LIN {X 0,Y 418.26,Z 369.386,A -85,B 0,C 180,E1 -10225.419,E2 -10225.419} C_VEL
LIN {X 0,Y 418.209,Z 369.388,A -85,B 0,C 180,E1 -10228.604,E2 -10228.604} C_VEL
LIN {X 0,Y 418.288,Z 369.379,A -85,B 0,C 180,E1 -10231.937,E2 -10231.937} C_VEL
LIN {X 0,Y 418.282,Z 369.366,A -85,B 0,C 180,E1 -10235.162,E2 -10235.162} C_VEL
LIN {X 0,Y 418.228,Z 369.385,A -85,B 0,C 180,E1 -10238.303,E2 -10238.303} C_VEL
LIN {X 0,Y 418.276,Z 369.382,A -85,B 0,C 180,E1 -10241.383,E2 -10241.383} C_VEL
LIN {X 0,Y 418.293,Z 369.376,A -85,B 0,C 180,E1 -10244.406,E2 -10244.406} C_VEL
LIN {X 0,Y 418.362,Z 369.372,A -85,B 0,C 180,E1 -10247.386,E2 -10247.386} C_VEL
LIN {X 0,Y 418.353,Z 369.367,A -85,B 0,C 180,E1 -10250.329,E2 -10250.329} C_VEL
LIN {X 0,Y 418.485,Z 369.352,A -85,B 0,C 180,E1 -10253.249,E2 -10253.249} C_VEL
LIN {X 0,Y 418.335,Z 369.376,A -85,B 0,C 180,E1 -10255.182,E2 -10255.182} C_VEL
LIN {X 0,Y 418.537,Z 369.345,A -85,B 0,C 180,E1 -10258.076,E2 -10258.076} C_VEL
LIN {X 0,Y 418.665,Z 369.329,A -85,B 0,C 180,E1 -10260,E2 -10260} C_VEL
LIN {X 0,Y 418.504,Z 369.351,A -85,B 0,C 180,E1 -10262.888,E2 -10262.888} C_VEL
LIN {X 0,Y 418.485,Z 369.357,A -85,B 0,C 180,E1 -10266.751,E2 -10266.751} C_VEL
LIN {X 0,Y 418.334,Z 369.372,A -85,B 0,C 180,E1 -10269.672,E2 -10269.672} C_VEL
LIN {X 0,Y 418.338,Z 369.373,A -85,B 0,C 180,E1 -10273.001,E2 -10273.001} C_VEL
LIN {X 0,Y 418.305,Z 369.376,A -85,B 0,C 180,E1 -10276.736,E2 -10276.736} C_VEL
LIN {X 0,Y 418.264,Z 369.382,A -85,B 0,C 180,E1 -10279.791,E2 -10279.791} C_VEL
LIN {X 0,Y 418.231,Z 369.389,A -85,B 0,C 180,E1 -10282.737,E2 -10282.737} C_VEL
LIN {X 0,Y 418.265,Z 369.372,A -85,B 0,C 180,E1 -10285.905,E2 -10285.905} C_VEL
LIN {X 0,Y 418.259,Z 369.382,A -85,B 0,C 180,E1 -10289.163,E2 -10289.163} C_VEL
LIN {X 0,Y 418.253,Z 369.384,A -85,B 0,C 180,E1 -10292.845,E2 -10292.845} C_VEL
LIN {X 0,Y 418.245,Z 369.388,A -85,B 0,C 180,E1 -10296.24,E2 -10296.24} C_VEL
LIN {X 0,Y 418.262,Z 369.384,A -85,B 0,C 180,E1 -10299.681,E2 -10299.681} C_VEL
LIN {X 0,Y 418.283,Z 369.379,A -85,B 0,C 180,E1 -10302.331,E2 -10302.331} C_VEL
LIN {X 0,Y 418.249,Z 369.388,A -85,B 0,C 180,E1 -10305.112,E2 -10305.112} C_VEL
LIN {X 0,Y 418.255,Z 369.391,A -85,B 0,C 180,E1 -10307.77,E2 -10307.77} C_VEL
LIN {X 0,Y 418.269,Z 369.384,A -85,B 0,C 180,E1 -10310.618,E2 -10310.618} C_VEL
LIN {X 0,Y 418.247,Z 369.387,A -85,B 0,C 180,E1 -10313.977,E2 -10313.977} C_VEL
LIN {X 0,Y 418.259,Z 369.385,A -85,B 0,C 180,E1 -10317.157,E2 -10317.157} C_VEL
LIN {X 0,Y 418.258,Z 369.391,A -85,B 0,C 180,E1 -10318.609,E2 -10318.609} C_VEL
LIN {X 0,Y 420.005,Z 378.049,A -85,B 0,C 180,E1 -10320.971,E2 -10320.971} C_VEL
LIN {X 0,Y 420.348,Z 380.959,A -85,B 0,C 180,E1 -10321.697,E2 -10321.697} C_VEL
LIN {X 0,Y 424.539,Z 397.902,A -85,B 0,C 180,E1 -10322.229,E2 -10322.229} C_VEL
LIN {X 0,Y 424.864,Z 400.946,A -85,B 0,C 180,E1 -10322.301,E2 -10322.301} C_VEL
LIN {X 0,Y 423.647,Z 487.611,A -85,B 0,C 180,E1 -10323.807,E2 -10323.807} C_VEL
LIN {X 0,Y 423.268,Z 499.777,A -85,B 0,C 180,E1 -10324.192,E2 -10324.192} C_VEL
LIN {X 0,Y 422.734,Z 512.426,A -85,B 0,C 180,E1 -10324.786,E2 -10324.786} C_VEL
LIN {X 0,Y 422.09,Z 524.174,A -85,B 0,C 180,E1 -10325.533,E2 -10325.533} C_VEL
LIN {X 0,Y 421.469,Z 534.802,A -85,B 0,C 180,E1 -10326.41,E2 -10326.41} C_VEL
LIN {X 0,Y 420.588,Z 545.68,A -85,B 0,C 180,E1 -10327.528,E2 -10327.528} C_VEL
LIN {X 0,Y 419.878,Z 554.518,A -85,B 0,C 180,E1 -10328.651,E2 -10328.651} C_VEL
LIN {X 0,Y 419.136,Z 563.264,A -85,B 0,C 180,E1 -10330.012,E2 -10330.012} C_VEL
LIN {X 0,Y 418.499,Z 570.426,A -85,B 0,C 180,E1 -10331.394,E2 -10331.394} C_VEL
LIN {X 0,Y 418.044,Z 576.652,A -85,B 0,C 180,E1 -10332.891,E2 -10332.891} C_VEL
LIN {X 0,Y 417.672,Z 581.55,A -85,B 0,C 180,E1 -10334.382,E2 -10334.382} C_VEL
LIN {X 0,Y 417.384,Z 585.282,A -85,B 0,C 180,E1 -10335.868,E2 -10335.868} C_VEL
LIN {X 0,Y 417.187,Z 588.485,A -85,B 0,C 180,E1 -10337.711,E2 -10337.711} C_VEL
LIN {X 0,Y 417.02,Z 590.19,A -85,B 0,C 180,E1 -10339.681,E2 -10339.681} C_VEL
LIN {X 0,Y 417.041,Z 590.444,A -85,B 0,C 180,E1 -10341.277,E2 -10341.277} C_VEL
LIN {X 0,Y 417.073,Z 590.067,A -85,B 0,C 180,E1 -10342.253,E2 -10342.253} C_VEL
LIN {X 0,Y 417.179,Z 588.496,A -85,B 0,C 180,E1 -10343.879,E2 -10343.879} C_VEL
LIN {X 0,Y 416.541,Z 587.399,A -85,B 0,C 180,E1 -10344.671,E2 -10344.671} C_VEL
LIN {X 0,Y 413.794,Z 585.076,A -85,B 0,C 180,E1 -10345.947,E2 -10345.947} C_VEL
LIN {X 0,Y 411.494,Z 582.788,A -85,B 0,C 180,E1 -10346.958,E2 -10346.958} C_VEL
LIN {X 0,Y 410.538,Z 580.679,A -85,B 0,C 180,E1 -10347.721,E2 -10347.721} C_VEL
LIN {X 0,Y 410.478,Z 579.858,A -85,B 0,C 180,E1 -10347.976,E2 -10347.976} C_VEL
LIN {X 0,Y 410.804,Z 574.307,A -85,B 0,C 180,E1 -10349.51,E2 -10349.51} C_VEL
LIN {X 0,Y 411.35,Z 567.599,A -85,B 0,C 180,E1 -10350.979,E2 -10350.979} C_VEL
LIN {X 0,Y 411.934,Z 559.285,A -85,B 0,C 180,E1 -10352.444,E2 -10352.444} C_VEL
LIN {X 0,Y 412.515,Z 550.731,A -85,B 0,C 180,E1 -10353.663,E2 -10353.663} C_VEL
LIN {X 0,Y 413.181,Z 540.216,A -85,B 0,C 180,E1 -10354.879,E2 -10354.879} C_VEL
LIN {X 0,Y 413.928,Z 529.748,A -85,B 0,C 180,E1 -10355.847,E2 -10355.847} C_VEL
LIN {X 0,Y 414.57,Z 518.155,A -85,B 0,C 180,E1 -10356.693,E2 -10356.693} C_VEL
LIN {X 0,Y 414.97,Z 506.184,A -85,B 0,C 180,E1 -10357.358,E2 -10357.358} C_VEL
LIN {X 0,Y 415.398,Z 493.099,A -85,B 0,C 180,E1 -10357.87,E2 -10357.87} C_VEL
LIN {X 0,Y 415.708,Z 480.345,A -85,B 0,C 180,E1 -10358.17,E2 -10358.17} C_VEL
LIN {X 0,Y 416.645,Z 399.493,A -85,B 0,C 180,E1 -10359.559,E2 -10359.559} C_VEL
LIN {X 0,Y 412.816,Z 380.72,A -85,B 0,C 180,E1 -10360.074,E2 -10360.074} C_VEL
LIN {X 0,Y 412.021,Z 373.906,A -85,B 0,C 180,E1 -10361.811,E2 -10361.811} C_VEL
LIN {X 0,Y 411.319,Z 370.252,A -85,B 0,C 180,E1 -10362.834,E2 -10362.834} C_VEL
LIN {X 0,Y 411.268,Z 370.259,A -85,B 0,C 180,E1 -10365.867,E2 -10365.867} C_VEL
LIN {X 0,Y 411.229,Z 370.259,A -85,B 0,C 180,E1 -10368.948,E2 -10368.948} C_VEL
LIN {X 0,Y 411.208,Z 370.263,A -85,B 0,C 180,E1 -10372.642,E2 -10372.642} C_VEL
LIN {X 0,Y 411.239,Z 370.256,A -85,B 0,C 180,E1 -10375.292,E2 -10375.292} C_VEL
LIN {X 0,Y 411.227,Z 370.261,A -85,B 0,C 180,E1 -10378.589,E2 -10378.589} C_VEL
LIN {X 0,Y 411.169,Z 370.268,A -85,B 0,C 180,E1 -10381.996,E2 -10381.996} C_VEL
LIN {X 0,Y 411.212,Z 370.262,A -85,B 0,C 180,E1 -10384.878,E2 -10384.878} C_VEL
LIN {X 0,Y 411.21,Z 370.265,A -85,B 0,C 180,E1 -10388.169,E2 -10388.169} C_VEL
LIN {X 0,Y 411.162,Z 370.267,A -85,B 0,C 180,E1 -10391.227,E2 -10391.227} C_VEL
LIN {X 0,Y 411.183,Z 370.267,A -85,B 0,C 180,E1 -10394.488,E2 -10394.488} C_VEL
LIN {X 0,Y 411.23,Z 370.258,A -85,B 0,C 180,E1 -10397.295,E2 -10397.295} C_VEL
LIN {X 0,Y 411.228,Z 370.261,A -85,B 0,C 180,E1 -10400.776,E2 -10400.776} C_VEL
LIN {X 0,Y 411.195,Z 370.265,A -85,B 0,C 180,E1 -10404.47,E2 -10404.47} C_VEL
LIN {X 0,Y 411.203,Z 370.263,A -85,B 0,C 180,E1 -10406.872,E2 -10406.872} C_VEL
LIN {X 0,Y 411.227,Z 370.261,A -85,B 0,C 180,E1 -10410.643,E2 -10410.643} C_VEL
LIN {X 0,Y 411.232,Z 370.259,A -85,B 0,C 180,E1 -10413.618,E2 -10413.618} C_VEL
LIN {X 0,Y 411.2,Z 370.263,A -85,B 0,C 180,E1 -10416.852,E2 -10416.852} C_VEL
LIN {X 0,Y 411.258,Z 370.258,A -85,B 0,C 180,E1 -10420.03,E2 -10420.03} C_VEL
LIN {X 0,Y 411.256,Z 370.256,A -85,B 0,C 180,E1 -10423.13,E2 -10423.13} C_VEL
LIN {X 0,Y 411.306,Z 370.25,A -85,B 0,C 180,E1 -10426.89,E2 -10426.89} C_VEL
LIN {X 0,Y 411.301,Z 370.252,A -85,B 0,C 180,E1 -10430.161,E2 -10430.161} C_VEL
LIN {X 0,Y 411.452,Z 370.231,A -85,B 0,C 180,E1 -10433.133,E2 -10433.133} C_VEL
LIN {X 0,Y 411.305,Z 370.249,A -85,B 0,C 180,E1 -10435.099,E2 -10435.099} C_VEL
LIN {X 0,Y 411.506,Z 370.227,A -85,B 0,C 180,E1 -10438.042,E2 -10438.042} C_VEL
LIN {X 0,Y 411.635,Z 370.211,A -85,B 0,C 180,E1 -10440,E2 -10440} C_VEL
LIN {X 0,Y 411.46,Z 370.23,A -85,B 0,C 180,E1 -10442.937,E2 -10442.937} C_VEL
LIN {X 0,Y 411.453,Z 370.231,A -85,B 0,C 180,E1 -10446.867,E2 -10446.867} C_VEL
LIN {X 0,Y 411.301,Z 370.252,A -85,B 0,C 180,E1 -10449.838,E2 -10449.838} C_VEL
LIN {X 0,Y 411.306,Z 370.249,A -85,B 0,C 180,E1 -10453.109,E2 -10453.109} C_VEL
LIN {X 0,Y 411.249,Z 370.256,A -85,B 0,C 180,E1 -10456.889,E2 -10456.889} C_VEL
LIN {X 0,Y 411.247,Z 370.259,A -85,B 0,C 180,E1 -10459.986,E2 -10459.986} C_VEL
LIN {X 0,Y 411.198,Z 370.262,A -85,B 0,C 180,E1 -10463.148,E2 -10463.148} C_VEL
LIN {X 0,Y 411.231,Z 370.261,A -85,B 0,C 180,E1 -10466.381,E2 -10466.381} C_VEL
LIN {X 0,Y 411.193,Z 370.265,A -85,B 0,C 180,E1 -10469.713,E2 -10469.713} C_VEL
LIN {X 0,Y 411.2,Z 370.262,A -85,B 0,C 180,E1 -10473.156,E2 -10473.156} C_VEL
LIN {X 0,Y 411.19,Z 370.264,A -85,B 0,C 180,E1 -10476.554,E2 -10476.554} C_VEL
LIN {X 0,Y 411.223,Z 370.262,A -85,B 0,C 180,E1 -10479.731,E2 -10479.731} C_VEL
LIN {X 0,Y 411.226,Z 370.258,A -85,B 0,C 180,E1 -10483.127,E2 -10483.127} C_VEL
LIN {X 0,Y 411.168,Z 370.27,A -85,B 0,C 180,E1 -10485.881,E2 -10485.881} C_VEL
LIN {X 0,Y 411.16,Z 370.266,A -85,B 0,C 180,E1 -10488.772,E2 -10488.772} C_VEL
LIN {X 0,Y 411.196,Z 370.266,A -85,B 0,C 180,E1 -10492.028,E2 -10492.028} C_VEL
LIN {X 0,Y 411.205,Z 370.264,A -85,B 0,C 180,E1 -10495.667,E2 -10495.667} C_VEL
LIN {X 0,Y 411.199,Z 370.262,A -85,B 0,C 180,E1 -10499.154,E2 -10499.154} C_VEL
LIN {X 0,Y 411.29,Z 370.439,A -85,B 0,C 180,E1 -10501.834,E2 -10501.834} C_VEL
LIN {X 0,Y 413.861,Z 383.381,A -85,B 0,C 180,E1 -10504.573,E2 -10504.573} C_VEL
LIN {X 0,Y 414.249,Z 387.672,A -85,B 0,C 180,E1 -10505.44,E2 -10505.44} C_VEL
LIN {X 0,Y 413.21,Z 403.81,A -85,B 0,C 180,E1 -10508.551,E2 -10508.551} C_VEL
LIN {X 0,Y 412.423,Z 416.273,A -85,B 0,C 180,E1 -10510.934,E2 -10510.934} C_VEL
LIN {X 0,Y 416.349,Z 445.438,A -85,B 0,C 180,E1 -10511.607,E2 -10511.607} C_VEL
LIN {X 0,Y 415.451,Z 525.237,A -85,B 0,C 180,E1 -10513.002,E2 -10513.002} C_VEL
LIN {X 0,Y 414.843,Z 539.187,A -85,B 0,C 180,E1 -10513.452,E2 -10513.452} C_VEL
LIN {X 0,Y 414.285,Z 551.698,A -85,B 0,C 180,E1 -10514.062,E2 -10514.062} C_VEL
LIN {X 0,Y 413.532,Z 563.64,A -85,B 0,C 180,E1 -10514.853,E2 -10514.853} C_VEL
LIN {X 0,Y 412.761,Z 575.122,A -85,B 0,C 180,E1 -10515.833,E2 -10515.833} C_VEL
LIN {X 0,Y 412.124,Z 585.675,A -85,B 0,C 180,E1 -10516.965,E2 -10516.965} C_VEL
LIN {X 0,Y 411.501,Z 594.764,A -85,B 0,C 180,E1 -10518.174,E2 -10518.174} C_VEL
LIN {X 0,Y 410.818,Z 603.786,A -85,B 0,C 180,E1 -10519.652,E2 -10519.652} C_VEL
LIN {X 0,Y 410.456,Z 611.054,A -85,B 0,C 180,E1 -10521.136,E2 -10521.136} C_VEL
LIN {X 0,Y 410.183,Z 616.842,A -85,B 0,C 180,E1 -10522.617,E2 -10522.617} C_VEL
LIN {X 0,Y 410.007,Z 621.393,A -85,B 0,C 180,E1 -10524.097,E2 -10524.097} C_VEL
LIN {X 0,Y 410.047,Z 623.795,A -85,B 0,C 180,E1 -10525.084,E2 -10525.084} C_VEL
LIN {X 0,Y 409.954,Z 625.753,A -85,B 0,C 180,E1 -10526.068,E2 -10526.068} C_VEL
LIN {X 0,Y 410.007,Z 627.296,A -85,B 0,C 180,E1 -10527.052,E2 -10527.052} C_VEL
LIN {X 0,Y 410.021,Z 628.38,A -85,B 0,C 180,E1 -10528.035,E2 -10528.035} C_VEL
LIN {X 0,Y 409.972,Z 629.348,A -85,B 0,C 180,E1 -10530,E2 -10530} C_VEL
LIN {X 0,Y 409.978,Z 629.25,A -85,B 0,C 180,E1 -10530.982,E2 -10530.982} C_VEL
LIN {X 0,Y 410.018,Z 628.721,A -85,B 0,C 180,E1 -10531.965,E2 -10531.965} C_VEL
LIN {X 0,Y 409.97,Z 627.786,A -85,B 0,C 180,E1 -10532.948,E2 -10532.948} C_VEL
LIN {X 0,Y 410.024,Z 624.725,A -85,B 0,C 180,E1 -10534.916,E2 -10534.916} C_VEL
LIN {X 0,Y 410.041,Z 621.689,A -85,B 0,C 180,E1 -10536.224,E2 -10536.224} C_VEL
LIN {X 0,Y 410.285,Z 616.703,A -85,B 0,C 180,E1 -10537.876,E2 -10537.876} C_VEL
LIN {X 0,Y 410.705,Z 609.834,A -85,B 0,C 180,E1 -10539.604,E2 -10539.604} C_VEL
LIN {X 0,Y 411.27,Z 602.404,A -85,B 0,C 180,E1 -10541.084,E2 -10541.084} C_VEL
LIN {X 0,Y 412.095,Z 593.192,A -85,B 0,C 180,E1 -10542.559,E2 -10542.559} C_VEL
LIN {X 0,Y 412.78,Z 583.641,A -85,B 0,C 180,E1 -10543.79,E2 -10543.79} C_VEL
LIN {X 0,Y 413.627,Z 573.075,A -85,B 0,C 180,E1 -10544.891,E2 -10544.891} C_VEL
LIN {X 0,Y 414.603,Z 561.291,A -85,B 0,C 180,E1 -10545.863,E2 -10545.863} C_VEL
LIN {X 0,Y 415.447,Z 548.69,A -85,B 0,C 180,E1 -10546.65,E2 -10546.65} C_VEL
LIN {X 0,Y 416.229,Z 535.368,A -85,B 0,C 180,E1 -10547.25,E2 -10547.25} C_VEL
LIN {X 0,Y 416.706,Z 523.005,A -85,B 0,C 180,E1 -10547.609,E2 -10547.609} C_VEL
LIN {X 0,Y 417.673,Z 444.319,A -85,B 0,C 180,E1 -10548.995,E2 -10548.995} C_VEL
LIN {X 0,Y 413.987,Z 421.068,A -85,B 0,C 180,E1 -10549.618,E2 -10549.618} C_VEL
LIN {X 0,Y 413.043,Z 415.819,A -85,B 0,C 180,E1 -10549.791,E2 -10549.791} C_VEL
LIN {X 0,Y 414.399,Z 397.757,A -85,B 0,C 180,E1 -10553.343,E2 -10553.343} C_VEL
LIN {X 0,Y 415.069,Z 389.228,A -85,B 0,C 180,E1 -10555.043,E2 -10555.043} C_VEL
LIN {X 0,Y 413.772,Z 381.411,A -85,B 0,C 180,E1 -10556.75,E2 -10556.75} C_VEL
LIN {X 0,Y 411.233,Z 370.258,A -85,B 0,C 180,E1 -10559.321,E2 -10559.321} C_VEL
LIN {X 0,Y 411.206,Z 370.263,A -85,B 0,C 180,E1 -10563.126,E2 -10563.126} C_VEL
LIN {X 0,Y 411.193,Z 370.265,A -85,B 0,C 180,E1 -10566.552,E2 -10566.552} C_VEL
LIN {X 0,Y 411.215,Z 370.263,A -85,B 0,C 180,E1 -10569.728,E2 -10569.728} C_VEL
LIN {X 0,Y 411.169,Z 370.264,A -85,B 0,C 180,E1 -10573.133,E2 -10573.133} C_VEL
LIN {X 0,Y 411.228,Z 370.259,A -85,B 0,C 180,E1 -10575.871,E2 -10575.871} C_VEL
LIN {X 0,Y 411.205,Z 370.257,A -85,B 0,C 180,E1 -10578.764,E2 -10578.764} C_VEL
LIN {X 0,Y 411.198,Z 370.261,A -85,B 0,C 180,E1 -10582.027,E2 -10582.027} C_VEL
LIN {X 0,Y 411.2,Z 370.265,A -85,B 0,C 180,E1 -10585.666,E2 -10585.666} C_VEL
LIN {X 0,Y 411.191,Z 370.266,A -85,B 0,C 180,E1 -10589.153,E2 -10589.153} C_VEL
LIN {X 0,Y 411.253,Z 370.254,A -85,B 0,C 180,E1 -10592.522,E2 -10592.522} C_VEL
LIN {X 0,Y 411.22,Z 370.249,A -85,B 0,C 180,E1 -10595.784,E2 -10595.784} C_VEL
LIN {X 0,Y 411.19,Z 370.265,A -85,B 0,C 180,E1 -10598.966,E2 -10598.966} C_VEL
LIN {X 0,Y 411.244,Z 370.255,A -85,B 0,C 180,E1 -10602.085,E2 -10602.085} C_VEL
LIN {X 0,Y 411.254,Z 370.254,A -85,B 0,C 180,E1 -10605.147,E2 -10605.147} C_VEL
LIN {X 0,Y 411.292,Z 370.249,A -85,B 0,C 180,E1 -10608.168,E2 -10608.168} C_VEL
LIN {X 0,Y 411.473,Z 370.227,A -85,B 0,C 180,E1 -10612.147,E2 -10612.147} C_VEL
LIN {X 0,Y 411.467,Z 370.222,A -85,B 0,C 180,E1 -10614.118,E2 -10614.118} C_VEL
LIN {X 0,Y 411.506,Z 370.221,A -85,B 0,C 180,E1 -10618.043,E2 -10618.043} C_VEL
LIN {X 0,Y 411.635,Z 370.205,A -85,B 0,C 180,E1 -10620,E2 -10620} C_VEL
LIN {X 0,Y 411.459,Z 370.228,A -85,B 0,C 180,E1 -10622.938,E2 -10622.938} C_VEL
LIN {X 0,Y 411.452,Z 370.231,A -85,B 0,C 180,E1 -10626.867,E2 -10626.867} C_VEL
LIN {X 0,Y 411.286,Z 370.25,A -85,B 0,C 180,E1 -10629.839,E2 -10629.839} C_VEL
LIN {X 0,Y 411.298,Z 370.249,A -85,B 0,C 180,E1 -10633.105,E2 -10633.105} C_VEL
LIN {X 0,Y 411.256,Z 370.254,A -85,B 0,C 180,E1 -10636.87,E2 -10636.87} C_VEL
LIN {X 0,Y 411.224,Z 370.26,A -85,B 0,C 180,E1 -10639.988,E2 -10639.988} C_VEL
LIN {X 0,Y 411.197,Z 370.262,A -85,B 0,C 180,E1 -10643.148,E2 -10643.148} C_VEL
LIN {X 0,Y 411.232,Z 370.245,A -85,B 0,C 180,E1 -10646.382,E2 -10646.382} C_VEL
LIN {X 0,Y 411.195,Z 370.263,A -85,B 0,C 180,E1 -10649.714,E2 -10649.714} C_VEL
LIN {X 0,Y 411.202,Z 370.261,A -85,B 0,C 180,E1 -10653.157,E2 -10653.157} C_VEL
LIN {X 0,Y 411.192,Z 370.264,A -85,B 0,C 180,E1 -10656.554,E2 -10656.554} C_VEL
LIN {X 0,Y 411.224,Z 370.262,A -85,B 0,C 180,E1 -10659.731,E2 -10659.731} C_VEL
LIN {X 0,Y 411.222,Z 370.259,A -85,B 0,C 180,E1 -10663.128,E2 -10663.128} C_VEL
LIN {X 0,Y 411.17,Z 370.269,A -85,B 0,C 180,E1 -10665.882,E2 -10665.882} C_VEL
LIN {X 0,Y 411.212,Z 370.267,A -85,B 0,C 180,E1 -10669.501,E2 -10669.501} C_VEL
LIN {X 0,Y 411.205,Z 370.266,A -85,B 0,C 180,E1 -10672.029,E2 -10672.029} C_VEL
LIN {X 0,Y 411.207,Z 370.264,A -85,B 0,C 180,E1 -10675.668,E2 -10675.668} C_VEL
LIN {X 0,Y 411.243,Z 370.437,A -85,B 0,C 180,E1 -10678.347,E2 -10678.347} C_VEL
LIN {X 0,Y 413.074,Z 379.492,A -85,B 0,C 180,E1 -10680.858,E2 -10680.858} C_VEL
LIN {X 0,Y 413.38,Z 381.416,A -85,B 0,C 180,E1 -10681.311,E2 -10681.311} C_VEL
LIN {X 0,Y 416.742,Z 393.57,A -85,B 0,C 180,E1 -10681.726,E2 -10681.726} C_VEL
LIN {X 0,Y 418.272,Z 401.497,A -85,B 0,C 180,E1 -10681.955,E2 -10681.955} C_VEL
LIN {X 0,Y 416.976,Z 487.866,A -85,B 0,C 180,E1 -10683.478,E2 -10683.478} C_VEL
LIN {X 0,Y 416.542,Z 500.63,A -85,B 0,C 180,E1 -10683.891,E2 -10683.891} C_VEL
LIN {X 0,Y 416.009,Z 512.932,A -85,B 0,C 180,E1 -10684.483,E2 -10684.483} C_VEL
LIN {X 0,Y 415.331,Z 524.629,A -85,B 0,C 180,E1 -10685.241,E2 -10685.241} C_VEL
LIN {X 0,Y 414.667,Z 535.319,A -85,B 0,C 180,E1 -10686.141,E2 -10686.141} C_VEL
LIN {X 0,Y 413.749,Z 546.088,A -85,B 0,C 180,E1 -10687.268,E2 -10687.268} C_VEL
LIN {X 0,Y 412.937,Z 555.815,A -85,B 0,C 180,E1 -10688.536,E2 -10688.536} C_VEL
LIN {X 0,Y 412.213,Z 563.693,A -85,B 0,C 180,E1 -10689.801,E2 -10689.801} C_VEL
LIN {X 0,Y 411.492,Z 571.362,A -85,B 0,C 180,E1 -10691.323,E2 -10691.323} C_VEL
LIN {X 0,Y 410.938,Z 578.382,A -85,B 0,C 180,E1 -10693.098,E2 -10693.098} C_VEL
LIN {X 0,Y 410.553,Z 582.966,A -85,B 0,C 180,E1 -10694.614,E2 -10694.614} C_VEL
LIN {X 0,Y 410.288,Z 586.419,A -85,B 0,C 180,E1 -10696.125,E2 -10696.125} C_VEL
LIN {X 0,Y 410.131,Z 588.831,A -85,B 0,C 180,E1 -10697.624,E2 -10697.624} C_VEL
LIN {X 0,Y 409.994,Z 590.297,A -85,B 0,C 180,E1 -10699.132,E2 -10699.132} C_VEL
LIN {X 0,Y 409.909,Z 590.756,A -85,B 0,C 180,E1 -10700.128,E2 -10700.128} C_VEL
LIN {X 0,Y 409.976,Z 590.459,A -85,B 0,C 180,E1 -10702.118,E2 -10702.118} C_VEL
LIN {X 0,Y 410.091,Z 588.842,A -85,B 0,C 180,E1 -10703.889,E2 -10703.889} C_VEL
LIN {X 0,Y 410.12,Z 587.009,A -85,B 0,C 180,E1 -10705.085,E2 -10705.085} C_VEL
LIN {X 0,Y 410.329,Z 583.857,A -85,B 0,C 180,E1 -10706.563,E2 -10706.563} C_VEL
LIN {X 0,Y 410.478,Z 579.858,A -85,B 0,C 180,E1 -10707.976,E2 -10707.976} C_VEL
LIN {X 0,Y 409.915,Z 577.429,A -85,B 0,C 180,E1 -10708.726,E2 -10708.726} C_VEL
LIN {X 0,Y 407.36,Z 573.051,A -85,B 0,C 180,E1 -10709.924,E2 -10709.924} C_VEL
LIN {X 0,Y 404.927,Z 568.02,A -85,B 0,C 180,E1 -10711.082,E2 -10711.082} C_VEL
LIN {X 0,Y 404.556,Z 564.541,A -85,B 0,C 180,E1 -10711.758,E2 -10711.758} C_VEL
LIN {X 0,Y 405.245,Z 555.484,A -85,B 0,C 180,E1 -10713.231,E2 -10713.231} C_VEL
LIN {X 0,Y 405.972,Z 544.95,A -85,B 0,C 180,E1 -10714.592,E2 -10714.592} C_VEL
LIN {X 0,Y 406.736,Z 534.195,A -85,B 0,C 180,E1 -10715.702,E2 -10715.702} C_VEL
LIN {X 0,Y 407.404,Z 523.685,A -85,B 0,C 180,E1 -10716.562,E2 -10716.562} C_VEL
LIN {X 0,Y 407.922,Z 511.113,A -85,B 0,C 180,E1 -10717.362,E2 -10717.362} C_VEL
LIN {X 0,Y 408.397,Z 498.485,A -85,B 0,C 180,E1 -10717.944,E2 -10717.944} C_VEL
LIN {X 0,Y 408.737,Z 486.317,A -85,B 0,C 180,E1 -10718.31,E2 -10718.31} C_VEL
LIN {X 0,Y 409.873,Z 400.613,A -85,B 0,C 180,E1 -10719.818,E2 -10719.818} C_VEL
LIN {X 0,Y 405.82,Z 381.046,A -85,B 0,C 180,E1 -10720.364,E2 -10720.364} C_VEL
LIN {X 0,Y 404.625,Z 372.722,A -85,B 0,C 180,E1 -10722.539,E2 -10722.539} C_VEL
LIN {X 0,Y 404.277,Z 371.129,A -85,B 0,C 180,E1 -10722.997,E2 -10722.997} C_VEL
LIN {X 0,Y 404.232,Z 371.135,A -85,B 0,C 180,E1 -10726.151,E2 -10726.151} C_VEL
LIN {X 0,Y 404.17,Z 371.137,A -85,B 0,C 180,E1 -10729.292,E2 -10729.292} C_VEL
LIN {X 0,Y 404.159,Z 371.14,A -85,B 0,C 180,E1 -10732.833,E2 -10732.833} C_VEL
LIN {X 0,Y 404.187,Z 371.135,A -85,B 0,C 180,E1 -10735.766,E2 -10735.766} C_VEL
LIN {X 0,Y 404.201,Z 371.135,A -85,B 0,C 180,E1 -10737.999,E2 -10737.999} C_VEL
LIN {X 0,Y 404.144,Z 371.14,A -85,B 0,C 180,E1 -10741.558,E2 -10741.558} C_VEL
LIN {X 0,Y 404.186,Z 371.136,A -85,B 0,C 180,E1 -10745.015,E2 -10745.015} C_VEL
LIN {X 0,Y 404.157,Z 371.141,A -85,B 0,C 180,E1 -10748.756,E2 -10748.756} C_VEL
LIN {X 0,Y 404.121,Z 371.144,A -85,B 0,C 180,E1 -10751.599,E2 -10751.599} C_VEL
LIN {X 0,Y 404.151,Z 371.143,A -85,B 0,C 180,E1 -10754.522,E2 -10754.522} C_VEL
LIN {X 0,Y 404.208,Z 371.133,A -85,B 0,C 180,E1 -10757.304,E2 -10757.304} C_VEL
LIN {X 0,Y 404.166,Z 371.141,A -85,B 0,C 180,E1 -10759.954,E2 -10759.954} C_VEL
LIN {X 0,Y 404.137,Z 371.142,A -85,B 0,C 180,E1 -10763.123,E2 -10763.123} C_VEL
LIN {X 0,Y 404.141,Z 371.145,A -85,B 0,C 180,E1 -10766.187,E2 -10766.187} C_VEL
LIN {X 0,Y 404.14,Z 371.143,A -85,B 0,C 180,E1 -10769.714,E2 -10769.714} C_VEL
LIN {X 0,Y 404.19,Z 371.135,A -85,B 0,C 180,E1 -10773.122,E2 -10773.122} C_VEL
LIN {X 0,Y 404.165,Z 371.141,A -85,B 0,C 180,E1 -10776.425,E2 -10776.425} C_VEL
LIN {X 0,Y 404.199,Z 371.138,A -85,B 0,C 180,E1 -10779.868,E2 -10779.868} C_VEL
LIN {X 0,Y 404.209,Z 371.133,A -85,B 0,C 180,E1 -10782.992,E2 -10782.992} C_VEL
LIN {X 0,Y 404.259,Z 371.128,A -85,B 0,C 180,E1 -10786.788,E2 -10786.788} C_VEL
LIN {X 0,Y 404.264,Z 371.129,A -85,B 0,C 180,E1 -10789.988,E2 -10789.988} C_VEL
LIN {X 0,Y 404.403,Z 371.109,A -85,B 0,C 180,E1 -10793.012,E2 -10793.012} C_VEL
LIN {X 0,Y 404.277,Z 371.125,A -85,B 0,C 180,E1 -10795.013,E2 -10795.013} C_VEL
LIN {X 0,Y 404.475,Z 371.103,A -85,B 0,C 180,E1 -10798.008,E2 -10798.008} C_VEL
LIN {X 0,Y 404.605,Z 371.087,A -85,B 0,C 180,E1 -10800,E2 -10800} C_VEL
LIN {X 0,Y 404.417,Z 371.107,A -85,B 0,C 180,E1 -10802.988,E2 -10802.988} C_VEL
LIN {X 0,Y 404.404,Z 371.109,A -85,B 0,C 180,E1 -10806.987,E2 -10806.987} C_VEL
LIN {X 0,Y 404.264,Z 371.129,A -85,B 0,C 180,E1 -10810.011,E2 -10810.011} C_VEL
LIN {X 0,Y 404.258,Z 371.127,A -85,B 0,C 180,E1 -10813.211,E2 -10813.211} C_VEL
LIN {X 0,Y 404.208,Z 371.133,A -85,B 0,C 180,E1 -10817.007,E2 -10817.007} C_VEL
LIN {X 0,Y 404.193,Z 371.138,A -85,B 0,C 180,E1 -10820.35,E2 -10820.35} C_VEL
LIN {X 0,Y 404.164,Z 371.141,A -85,B 0,C 180,E1 -10823.575,E2 -10823.575} C_VEL
LIN {X 0,Y 404.188,Z 371.135,A -85,B 0,C 180,E1 -10826.878,E2 -10826.878} C_VEL
LIN {X 0,Y 404.138,Z 371.145,A -85,B 0,C 180,E1 -10830.286,E2 -10830.286} C_VEL
LIN {X 0,Y 404.139,Z 371.145,A -85,B 0,C 180,E1 -10833.813,E2 -10833.813} C_VEL
LIN {X 0,Y 404.135,Z 371.142,A -85,B 0,C 180,E1 -10836.876,E2 -10836.876} C_VEL
LIN {X 0,Y 404.163,Z 371.143,A -85,B 0,C 180,E1 -10840.084,E2 -10840.084} C_VEL
LIN {X 0,Y 404.2,Z 371.133,A -85,B 0,C 180,E1 -10843.092,E2 -10843.092} C_VEL
LIN {X 0,Y 404.147,Z 371.145,A -85,B 0,C 180,E1 -10845.927,E2 -10845.927} C_VEL
LIN {X 0,Y 404.114,Z 371.144,A -85,B 0,C 180,E1 -10848.636,E2 -10848.636} C_VEL
LIN {X 0,Y 404.153,Z 371.141,A -85,B 0,C 180,E1 -10851.492,E2 -10851.492} C_VEL
LIN {X 0,Y 404.183,Z 371.135,A -85,B 0,C 180,E1 -10854.985,E2 -10854.985} C_VEL
LIN {X 0,Y 404.148,Z 371.139,A -85,B 0,C 180,E1 -10858.555,E2 -10858.555} C_VEL
LIN {X 0,Y 404.238,Z 371.226,A -85,B 0,C 180,E1 -10861.58,E2 -10861.58} C_VEL
LIN {X 0,Y 406.506,Z 382.537,A -85,B 0,C 180,E1 -10864.029,E2 -10864.029} C_VEL
LIN {X 0,Y 407.304,Z 388.468,A -85,B 0,C 180,E1 -10865.265,E2 -10865.265} C_VEL
LIN {X 0,Y 406.207,Z 404.596,A -85,B 0,C 180,E1 -10868.429,E2 -10868.429} C_VEL
LIN {X 0,Y 405.462,Z 415.961,A -85,B 0,C 180,E1 -10870.641,E2 -10870.641} C_VEL
LIN {X 0,Y 409.518,Z 445.084,A -85,B 0,C 180,E1 -10871.332,E2 -10871.332} C_VEL
LIN {X 0,Y 408.595,Z 524.516,A -85,B 0,C 180,E1 -10872.74,E2 -10872.74} C_VEL
LIN {X 0,Y 408.044,Z 537.839,A -85,B 0,C 180,E1 -10873.168,E2 -10873.168} C_VEL
LIN {X 0,Y 407.415,Z 550.633,A -85,B 0,C 180,E1 -10873.786,E2 -10873.786} C_VEL
LIN {X 0,Y 406.661,Z 562.784,A -85,B 0,C 180,E1 -10874.591,E2 -10874.591} C_VEL
LIN {X 0,Y 405.807,Z 574.358,A -85,B 0,C 180,E1 -10875.585,E2 -10875.585} C_VEL
LIN {X 0,Y 405.153,Z 585.264,A -85,B 0,C 180,E1 -10876.769,E2 -10876.769} C_VEL
LIN {X 0,Y 404.522,Z 594.164,A -85,B 0,C 180,E1 -10877.967,E2 -10877.967} C_VEL
LIN {X 0,Y 403.793,Z 603.232,A -85,B 0,C 180,E1 -10879.47,E2 -10879.47} C_VEL
LIN {X 0,Y 403.379,Z 610.541,A -85,B 0,C 180,E1 -10880.979,E2 -10880.979} C_VEL
LIN {X 0,Y 403.129,Z 616.378,A -85,B 0,C 180,E1 -10882.487,E2 -10882.487} C_VEL
LIN {X 0,Y 402.938,Z 620.961,A -85,B 0,C 180,E1 -10883.993,E2 -10883.993} C_VEL
LIN {X 0,Y 402.954,Z 623.378,A -85,B 0,C 180,E1 -10884.997,E2 -10884.997} C_VEL
LIN {X 0,Y 402.874,Z 625.35,A -85,B 0,C 180,E1 -10885.999,E2 -10885.999} C_VEL
LIN {X 0,Y 402.906,Z 626.909,A -85,B 0,C 180,E1 -10887,E2 -10887} C_VEL
LIN {X 0,Y 402.951,Z 628.016,A -85,B 0,C 180,E1 -10888.001,E2 -10888.001} C_VEL
LIN {X 0,Y 402.894,Z 629.008,A -85,B 0,C 180,E1 -10890,E2 -10890} C_VEL
LIN {X 0,Y 402.903,Z 628.924,A -85,B 0,C 180,E1 -10890.999,E2 -10890.999} C_VEL
LIN {X 0,Y 402.946,Z 628.419,A -85,B 0,C 180,E1 -10891.999,E2 -10891.999} C_VEL
LIN {X 0,Y 402.861,Z 626.179,A -85,B 0,C 180,E1 -10894.001,E2 -10894.001} C_VEL
LIN {X 0,Y 402.92,Z 623.404,A -85,B 0,C 180,E1 -10895.505,E2 -10895.505} C_VEL
LIN {X 0,Y 403.076,Z 619.614,A -85,B 0,C 180,E1 -10897.01,E2 -10897.01} C_VEL
LIN {X 0,Y 403.328,Z 614.712,A -85,B 0,C 180,E1 -10898.517,E2 -10898.517} C_VEL
LIN {X 0,Y 403.746,Z 608.555,A -85,B 0,C 180,E1 -10900.024,E2 -10900.024} C_VEL
LIN {X 0,Y 404.387,Z 600.926,A -85,B 0,C 180,E1 -10901.529,E2 -10901.529} C_VEL
LIN {X 0,Y 405.156,Z 593.143,A -85,B 0,C 180,E1 -10902.777,E2 -10902.777} C_VEL
LIN {X 0,Y 405.862,Z 583.662,A -85,B 0,C 180,E1 -10904.03,E2 -10904.03} C_VEL
LIN {X 0,Y 406.78,Z 573.173,A -85,B 0,C 180,E1 -10905.148,E2 -10905.148} C_VEL
LIN {X 0,Y 407.77,Z 561.524,A -85,B 0,C 180,E1 -10906.136,E2 -10906.136} C_VEL
LIN {X 0,Y 408.687,Z 549.117,A -85,B 0,C 180,E1 -10906.933,E2 -10906.933} C_VEL
LIN {X 0,Y 409.482,Z 536.076,A -85,B 0,C 180,E1 -10907.543,E2 -10907.543} C_VEL
LIN {X 0,Y 410.017,Z 523.226,A -85,B 0,C 180,E1 -10907.938,E2 -10907.938} C_VEL
LIN {X 0,Y 410.998,Z 444.67,A -85,B 0,C 180,E1 -10909.349,E2 -10909.349} C_VEL
LIN {X 0,Y 407.41,Z 422.07,A -85,B 0,C 180,E1 -10909.971,E2 -10909.971} C_VEL
LIN {X 0,Y 406.164,Z 415.444,A -85,B 0,C 180,E1 -10910.196,E2 -10910.196} C_VEL
LIN {X 0,Y 407.437,Z 399.584,A -85,B 0,C 180,E1 -10913.374,E2 -10913.374} C_VEL
LIN {X 0,Y 408.187,Z 390.47,A -85,B 0,C 180,E1 -10915.222,E2 -10915.222} C_VEL
LIN {X 0,Y 406.564,Z 381.37,A -85,B 0,C 180,E1 -10917.263,E2 -10917.263} C_VEL
LIN {X 0,Y 404.177,Z 371.137,A -85,B 0,C 180,E1 -10919.705,E2 -10919.705} C_VEL
LIN {X 0,Y 404.169,Z 371.14,A -85,B 0,C 180,E1 -10923.419,E2 -10923.419} C_VEL
LIN {X 0,Y 404.142,Z 371.145,A -85,B 0,C 180,E1 -10926.245,E2 -10926.245} C_VEL
LIN {X 0,Y 404.156,Z 371.139,A -85,B 0,C 180,E1 -10928.756,E2 -10928.756} C_VEL
LIN {X 0,Y 404.12,Z 371.145,A -85,B 0,C 180,E1 -10931.599,E2 -10931.599} C_VEL
LIN {X 0,Y 404.149,Z 371.137,A -85,B 0,C 180,E1 -10934.523,E2 -10934.523} C_VEL
LIN {X 0,Y 404.204,Z 371.132,A -85,B 0,C 180,E1 -10937.304,E2 -10937.304} C_VEL
LIN {X 0,Y 404.164,Z 371.139,A -85,B 0,C 180,E1 -10939.955,E2 -10939.955} C_VEL
LIN {X 0,Y 404.135,Z 371.141,A -85,B 0,C 180,E1 -10943.124,E2 -10943.124} C_VEL
LIN {X 0,Y 404.139,Z 371.141,A -85,B 0,C 180,E1 -10946.187,E2 -10946.187} C_VEL
LIN {X 0,Y 404.147,Z 371.141,A -85,B 0,C 180,E1 -10949.715,E2 -10949.715} C_VEL
LIN {X 0,Y 404.189,Z 371.134,A -85,B 0,C 180,E1 -10953.123,E2 -10953.123} C_VEL
LIN {X 0,Y 404.17,Z 371.123,A -85,B 0,C 180,E1 -10955.334,E2 -10955.334} C_VEL
LIN {X 0,Y 404.132,Z 371.142,A -85,B 0,C 180,E1 -10958.58,E2 -10958.58} C_VEL
LIN {X 0,Y 404.202,Z 371.134,A -85,B 0,C 180,E1 -10961.762,E2 -10961.762} C_VEL
LIN {X 0,Y 404.199,Z 371.133,A -85,B 0,C 180,E1 -10964.882,E2 -10964.882} C_VEL
LIN {X 0,Y 404.263,Z 371.125,A -85,B 0,C 180,E1 -10967.959,E2 -10967.959} C_VEL
LIN {X 0,Y 404.425,Z 371.105,A -85,B 0,C 180,E1 -10972.1,E2 -10972.1} C_VEL
LIN {X 0,Y 404.415,Z 371.1,A -85,B 0,C 180,E1 -10974.015,E2 -10974.015} C_VEL
LIN {X 0,Y 404.475,Z 371.096,A -85,B 0,C 180,E1 -10978.009,E2 -10978.009} C_VEL
LIN {X 0,Y 404.605,Z 371.081,A -85,B 0,C 180,E1 -10980,E2 -10980} C_VEL
LIN {X 0,Y 404.416,Z 371.104,A -85,B 0,C 180,E1 -10982.989,E2 -10982.989} C_VEL
LIN {X 0,Y 404.399,Z 371.108,A -85,B 0,C 180,E1 -10986.988,E2 -10986.988} C_VEL
LIN {X 0,Y 404.251,Z 371.127,A -85,B 0,C 180,E1 -10990.012,E2 -10990.012} C_VEL
LIN {X 0,Y 404.259,Z 371.125,A -85,B 0,C 180,E1 -10993.212,E2 -10993.212} C_VEL
LIN {X 0,Y 404.209,Z 371.131,A -85,B 0,C 180,E1 -10997.008,E2 -10997.008} C_VEL
LIN {X 0,Y 404.157,Z 371.141,A -85,B 0,C 180,E1 -11000.352,E2 -11000.352} C_VEL
LIN {X 0,Y 404.163,Z 371.138,A -85,B 0,C 180,E1 -11003.575,E2 -11003.575} C_VEL
LIN {X 0,Y 404.178,Z 371.127,A -85,B 0,C 180,E1 -11005.767,E2 -11005.767} C_VEL
LIN {X 0,Y 404.19,Z 371.129,A -85,B 0,C 180,E1 -11008.001,E2 -11008.001} C_VEL
LIN {X 0,Y 404.134,Z 371.139,A -85,B 0,C 180,E1 -11011.559,E2 -11011.559} C_VEL
LIN {X 0,Y 404.181,Z 371.137,A -85,B 0,C 180,E1 -11015.017,E2 -11015.017} C_VEL
LIN {X 0,Y 404.16,Z 371.139,A -85,B 0,C 180,E1 -11018.757,E2 -11018.757} C_VEL
LIN {X 0,Y 404.189,Z 371.139,A -85,B 0,C 180,E1 -11021.612,E2 -11021.612} C_VEL
LIN {X 0,Y 404.189,Z 371.141,A -85,B 0,C 180,E1 -11024.53,E2 -11024.53} C_VEL
LIN {X 0,Y 404.17,Z 371.142,A -85,B 0,C 180,E1 -11027.301,E2 -11027.301} C_VEL
LIN {X 0,Y 404.168,Z 371.144,A -85,B 0,C 180,E1 -11029.956,E2 -11029.956} C_VEL
LIN {X 0,Y 404.141,Z 371.144,A -85,B 0,C 180,E1 -11033.125,E2 -11033.125} C_VEL
LIN {X 0,Y 404.146,Z 371.145,A -85,B 0,C 180,E1 -11036.189,E2 -11036.189} C_VEL
LIN {X 0,Y 404.186,Z 371.262,A -85,B 0,C 180,E1 -11038.013,E2 -11038.013} C_VEL
LIN {X 0,Y 405.951,Z 379.844,A -85,B 0,C 180,E1 -11040.437,E2 -11040.437} C_VEL
LIN {X 0,Y 406.298,Z 381.73,A -85,B 0,C 180,E1 -11040.9,E2 -11040.9} C_VEL
LIN {X 0,Y 408.971,Z 389.995,A -85,B 0,C 180,E1 -11041.214,E2 -11041.214} C_VEL
LIN {X 0,Y 411.641,Z 401.3,A -85,B 0,C 180,E1 -11041.579,E2 -11041.579} C_VEL
LIN {X 0,Y 410.332,Z 488.497,A -85,B 0,C 180,E1 -11043.148,E2 -11043.148} C_VEL
LIN {X 0,Y 409.878,Z 500.99,A -85,B 0,C 180,E1 -11043.56,E2 -11043.56} C_VEL
LIN {X 0,Y 409.303,Z 513.468,A -85,B 0,C 180,E1 -11044.17,E2 -11044.17} C_VEL
LIN {X 0,Y 408.586,Z 525.104,A -85,B 0,C 180,E1 -11044.94,E2 -11044.94} C_VEL
LIN {X 0,Y 407.878,Z 536,A -85,B 0,C 180,E1 -11045.878,E2 -11045.878} C_VEL
LIN {X 0,Y 406.932,Z 546.51,A -85,B 0,C 180,E1 -11046.999,E2 -11046.999} C_VEL
LIN {X 0,Y 406.133,Z 555.317,A -85,B 0,C 180,E1 -11048.158,E2 -11048.158} C_VEL
LIN {X 0,Y 405.396,Z 563.193,A -85,B 0,C 180,E1 -11049.417,E2 -11049.417} C_VEL
LIN {X 0,Y 404.578,Z 571.173,A -85,B 0,C 180,E1 -11050.992,E2 -11050.992} C_VEL
LIN {X 0,Y 404.121,Z 576.465,A -85,B 0,C 180,E1 -11052.282,E2 -11052.282} C_VEL
LIN {X 0,Y 403.674,Z 581.546,A -85,B 0,C 180,E1 -11053.826,E2 -11053.826} C_VEL
LIN {X 0,Y 403.327,Z 585.448,A -85,B 0,C 180,E1 -11055.365,E2 -11055.365} C_VEL
LIN {X 0,Y 403.067,Z 589.186,A -85,B 0,C 180,E1 -11057.539,E2 -11057.539} C_VEL
LIN {X 0,Y 402.941,Z 590.538,A -85,B 0,C 180,E1 -11058.939,E2 -11058.939} C_VEL
LIN {X 0,Y 402.827,Z 591.068,A -85,B 0,C 180,E1 -11059.953,E2 -11059.953} C_VEL
LIN {X 0,Y 402.838,Z 591.154,A -85,B 0,C 180,E1 -11060.966,E2 -11060.966} C_VEL
LIN {X 0,Y 402.952,Z 590.162,A -85,B 0,C 180,E1 -11062.987,E2 -11062.987} C_VEL
LIN {X 0,Y 403.002,Z 589.078,A -85,B 0,C 180,E1 -11063.994,E2 -11063.994} C_VEL
LIN {X 0,Y 403.046,Z 587.549,A -85,B 0,C 180,E1 -11064.998,E2 -11064.998} C_VEL
LIN {X 0,Y 403.241,Z 584.478,A -85,B 0,C 180,E1 -11066.503,E2 -11066.503} C_VEL
LIN {X 0,Y 403.42,Z 580.338,A -85,B 0,C 180,E1 -11068.014,E2 -11068.014} C_VEL
LIN {X 0,Y 403.808,Z 574.105,A -85,B 0,C 180,E1 -11069.751,E2 -11069.751} C_VEL
LIN {X 0,Y 404.381,Z 567.278,A -85,B 0,C 180,E1 -11071.245,E2 -11071.245} C_VEL
LIN {X 0,Y 404.556,Z 564.541,A -85,B 0,C 180,E1 -11071.758,E2 -11071.758} C_VEL
LIN {X 0,Y 404.196,Z 560.886,A -85,B 0,C 180,E1 -11072.415,E2 -11072.415} C_VEL
LIN {X 0,Y 401.856,Z 554.683,A -85,B 0,C 180,E1 -11073.464,E2 -11073.464} C_VEL
LIN {X 0,Y 399.513,Z 547.945,A -85,B 0,C 180,E1 -11074.451,E2 -11074.451} C_VEL
LIN {X 0,Y 399.147,Z 543.453,A -85,B 0,C 180,E1 -11075,E2 -11075} C_VEL
LIN {X 0,Y 399.916,Z 532.999,A -85,B 0,C 180,E1 -11076.052,E2 -11076.052} C_VEL
LIN {X 0,Y 400.632,Z 522.106,A -85,B 0,C 180,E1 -11076.927,E2 -11076.927} C_VEL
LIN {X 0,Y 401.107,Z 510.122,A -85,B 0,C 180,E1 -11077.678,E2 -11077.678} C_VEL
LIN {X 0,Y 401.585,Z 497.648,A -85,B 0,C 180,E1 -11078.238,E2 -11078.238} C_VEL
LIN {X 0,Y 401.914,Z 484.622,A -85,B 0,C 180,E1 -11078.611,E2 -11078.611} C_VEL
LIN {X 0,Y 402.983,Z 401.199,A -85,B 0,C 180,E1 -11080.099,E2 -11080.099} C_VEL
LIN {X 0,Y 399.166,Z 383.034,A -85,B 0,C 180,E1 -11080.601,E2 -11080.601} C_VEL
LIN {X 0,Y 398.765,Z 381.323,A -85,B 0,C 180,E1 -11080.68,E2 -11080.68} C_VEL
LIN {X 0,Y 397.247,Z 372.004,A -85,B 0,C 180,E1 -11083.178,E2 -11083.178} C_VEL
LIN {X 0,Y 397.176,Z 372.014,A -85,B 0,C 180,E1 -11086.446,E2 -11086.446} C_VEL
LIN {X 0,Y 397.152,Z 372.011,A -85,B 0,C 180,E1 -11089.646,E2 -11089.646} C_VEL
LIN {X 0,Y 397.139,Z 372.013,A -85,B 0,C 180,E1 -11093.04,E2 -11093.04} C_VEL
LIN {X 0,Y 397.138,Z 372.018,A -85,B 0,C 180,E1 -11096.257,E2 -11096.257} C_VEL
LIN {X 0,Y 397.13,Z 372.018,A -85,B 0,C 180,E1 -11098.542,E2 -11098.542} C_VEL
LIN {X 0,Y 397.082,Z 372.023,A -85,B 0,C 180,E1 -11102.07,E2 -11102.07} C_VEL
LIN {X 0,Y 397.121,Z 372.015,A -85,B 0,C 180,E1 -11105.503,E2 -11105.503} C_VEL
LIN {X 0,Y 397.132,Z 372.016,A -85,B 0,C 180,E1 -11108.861,E2 -11108.861} C_VEL
LIN {X 0,Y 397.068,Z 372.027,A -85,B 0,C 180,E1 -11112.266,E2 -11112.266} C_VEL
LIN {X 0,Y 397.115,Z 372.016,A -85,B 0,C 180,E1 -11115.063,E2 -11115.063} C_VEL
LIN {X 0,Y 397.154,Z 372.015,A -85,B 0,C 180,E1 -11118.006,E2 -11118.006} C_VEL
LIN {X 0,Y 397.106,Z 372.019,A -85,B 0,C 180,E1 -11121.725,E2 -11121.725} C_VEL
LIN {X 0,Y 397.122,Z 372.016,A -85,B 0,C 180,E1 -11125.506,E2 -11125.506} C_VEL
LIN {X 0,Y 397.073,Z 372.022,A -85,B 0,C 180,E1 -11129.117,E2 -11129.117} C_VEL
LIN {X 0,Y 397.189,Z 372.01,A -85,B 0,C 180,E1 -11132.609,E2 -11132.609} C_VEL
LIN {X 0,Y 397.128,Z 372.019,A -85,B 0,C 180,E1 -11135.981,E2 -11135.981} C_VEL
LIN {X 0,Y 397.15,Z 372.014,A -85,B 0,C 180,E1 -11139.697,E2 -11139.697} C_VEL
LIN {X 0,Y 397.175,Z 372.01,A -85,B 0,C 180,E1 -11142.844,E2 -11142.844} C_VEL
LIN {X 0,Y 397.219,Z 372.005,A -85,B 0,C 180,E1 -11146.678,E2 -11146.678} C_VEL
LIN {X 0,Y 397.222,Z 372.006,A -85,B 0,C 180,E1 -11149.809,E2 -11149.809} C_VEL
LIN {X 0,Y 397.356,Z 371.987,A -85,B 0,C 180,E1 -11152.888,E2 -11152.888} C_VEL
LIN {X 0,Y 397.249,Z 372,A -85,B 0,C 180,E1 -11154.925,E2 -11154.925} C_VEL
LIN {X 0,Y 397.444,Z 371.979,A -85,B 0,C 180,E1 -11157.973,E2 -11157.973} C_VEL
LIN {X 0,Y 397.574,Z 371.963,A -85,B 0,C 180,E1 -11160,E2 -11160} C_VEL
LIN {X 0,Y 397.376,Z 371.984,A -85,B 0,C 180,E1 -11163.041,E2 -11163.041} C_VEL
LIN {X 0,Y 397.356,Z 371.986,A -85,B 0,C 180,E1 -11167.112,E2 -11167.112} C_VEL
LIN {X 0,Y 397.222,Z 372.007,A -85,B 0,C 180,E1 -11170.191,E2 -11170.191} C_VEL
LIN {X 0,Y 397.218,Z 372.004,A -85,B 0,C 180,E1 -11173.321,E2 -11173.321} C_VEL
LIN {X 0,Y 397.174,Z 372.009,A -85,B 0,C 180,E1 -11177.155,E2 -11177.155} C_VEL
LIN {X 0,Y 397.125,Z 372.016,A -85,B 0,C 180,E1 -11180.729,E2 -11180.729} C_VEL
LIN {X 0,Y 397.127,Z 372.019,A -85,B 0,C 180,E1 -11184.019,E2 -11184.019} C_VEL
LIN {X 0,Y 397.187,Z 372.008,A -85,B 0,C 180,E1 -11187.391,E2 -11187.391} C_VEL
LIN {X 0,Y 397.071,Z 372.021,A -85,B 0,C 180,E1 -11190.883,E2 -11190.883} C_VEL
LIN {X 0,Y 397.12,Z 372.017,A -85,B 0,C 180,E1 -11194.494,E2 -11194.494} C_VEL
LIN {X 0,Y 397.104,Z 372.02,A -85,B 0,C 180,E1 -11198.275,E2 -11198.275} C_VEL
LIN {X 0,Y 397.152,Z 372.017,A -85,B 0,C 180,E1 -11201.994,E2 -11201.994} C_VEL
LIN {X 0,Y 397.108,Z 372.017,A -85,B 0,C 180,E1 -11205.066,E2 -11205.066} C_VEL
LIN {X 0,Y 397.063,Z 372.027,A -85,B 0,C 180,E1 -11208.022,E2 -11208.022} C_VEL
LIN {X 0,Y 397.128,Z 372.014,A -85,B 0,C 180,E1 -11211.139,E2 -11211.139} C_VEL
LIN {X 0,Y 397.118,Z 372.016,A -85,B 0,C 180,E1 -11214.497,E2 -11214.497} C_VEL
LIN {X 0,Y 397.11,Z 372.022,A -85,B 0,C 180,E1 -11217.932,E2 -11217.932} C_VEL
LIN {X 0,Y 397.183,Z 372.167,A -85,B 0,C 180,E1 -11221.354,E2 -11221.354} C_VEL
LIN {X 0,Y 399.772,Z 385.135,A -85,B 0,C 180,E1 -11224.209,E2 -11224.209} C_VEL
LIN {X 0,Y 400.353,Z 389.251,A -85,B 0,C 180,E1 -11225.083,E2 -11225.083} C_VEL
LIN {X 0,Y 399.218,Z 405.36,A -85,B 0,C 180,E1 -11228.304,E2 -11228.304} C_VEL
LIN {X 0,Y 398.51,Z 415.629,A -85,B 0,C 180,E1 -11230.339,E2 -11230.339} C_VEL
LIN {X 0,Y 402.699,Z 446.434,A -85,B 0,C 180,E1 -11231.082,E2 -11231.082} C_VEL
LIN {X 0,Y 401.74,Z 523.708,A -85,B 0,C 180,E1 -11232.469,E2 -11232.469} C_VEL
LIN {X 0,Y 401.21,Z 537.219,A -85,B 0,C 180,E1 -11232.905,E2 -11232.905} C_VEL
LIN {X 0,Y 400.535,Z 549.512,A -85,B 0,C 180,E1 -11233.499,E2 -11233.499} C_VEL
LIN {X 0,Y 399.764,Z 561.903,A -85,B 0,C 180,E1 -11234.318,E2 -11234.318} C_VEL
LIN {X 0,Y 398.899,Z 573.58,A -85,B 0,C 180,E1 -11235.329,E2 -11235.329} C_VEL
LIN {X 0,Y 398.271,Z 583.406,A -85,B 0,C 180,E1 -11236.395,E2 -11236.395} C_VEL
LIN {X 0,Y 397.523,Z 593.552,A -85,B 0,C 180,E1 -11237.752,E2 -11237.752} C_VEL
LIN {X 0,Y 396.783,Z 602.67,A -85,B 0,C 180,E1 -11239.282,E2 -11239.282} C_VEL
LIN {X 0,Y 396.334,Z 610.021,A -85,B 0,C 180,E1 -11240.817,E2 -11240.817} C_VEL
LIN {X 0,Y 396.056,Z 615.902,A -85,B 0,C 180,E1 -11242.352,E2 -11242.352} C_VEL
LIN {X 0,Y 395.831,Z 621.276,A -85,B 0,C 180,E1 -11244.19,E2 -11244.19} C_VEL
LIN {X 0,Y 395.796,Z 624.944,A -85,B 0,C 180,E1 -11245.927,E2 -11245.927} C_VEL
LIN {X 0,Y 395.807,Z 626.516,A -85,B 0,C 180,E1 -11246.947,E2 -11246.947} C_VEL
LIN {X 0,Y 395.881,Z 627.651,A -85,B 0,C 180,E1 -11247.965,E2 -11247.965} C_VEL
LIN {X 0,Y 395.819,Z 628.669,A -85,B 0,C 180,E1 -11250,E2 -11250} C_VEL
LIN {X 0,Y 395.83,Z 628.597,A -85,B 0,C 180,E1 -11251.017,E2 -11251.017} C_VEL
LIN {X 0,Y 395.856,Z 628.117,A -85,B 0,C 180,E1 -11252.035,E2 -11252.035} C_VEL
LIN {X 0,Y 395.783,Z 625.903,A -85,B 0,C 180,E1 -11254.073,E2 -11254.073} C_VEL
LIN {X 0,Y 395.828,Z 622.724,A -85,B 0,C 180,E1 -11255.808,E2 -11255.808} C_VEL
LIN {X 0,Y 396.063,Z 617.92,A -85,B 0,C 180,E1 -11257.648,E2 -11257.648} C_VEL
LIN {X 0,Y 396.466,Z 611.634,A -85,B 0,C 180,E1 -11259.437,E2 -11259.437} C_VEL
LIN {X 0,Y 396.992,Z 604.813,A -85,B 0,C 180,E1 -11260.971,E2 -11260.971} C_VEL
LIN {X 0,Y 397.899,Z 596.356,A -85,B 0,C 180,E1 -11262.496,E2 -11262.496} C_VEL
LIN {X 0,Y 398.685,Z 586.592,A -85,B 0,C 180,E1 -11263.911,E2 -11263.911} C_VEL
LIN {X 0,Y 399.685,Z 575.953,A -85,B 0,C 180,E1 -11265.149,E2 -11265.149} C_VEL
LIN {X 0,Y 400.722,Z 564.903,A -85,B 0,C 180,E1 -11266.166,E2 -11266.166} C_VEL
LIN {X 0,Y 401.714,Z 552.677,A -85,B 0,C 180,E1 -11267.04,E2 -11267.04} C_VEL
LIN {X 0,Y 402.576,Z 539.832,A -85,B 0,C 180,E1 -11267.723,E2 -11267.723} C_VEL
LIN {X 0,Y 403.236,Z 526.87,A -85,B 0,C 180,E1 -11268.185,E2 -11268.185} C_VEL
LIN {X 0,Y 403.652,Z 507.912,A -85,B 0,C 180,E1 -11268.573,E2 -11268.573} C_VEL
LIN {X 0,Y 404.424,Z 445.698,A -85,B 0,C 180,E1 -11269.698,E2 -11269.698} C_VEL
LIN {X 0,Y 401.006,Z 423.955,A -85,B 0,C 180,E1 -11270.31,E2 -11270.31} C_VEL
LIN {X 0,Y 399.306,Z 415.101,A -85,B 0,C 180,E1 -11270.61,E2 -11270.61} C_VEL
LIN {X 0,Y 400.529,Z 400.818,A -85,B 0,C 180,E1 -11273.527,E2 -11273.527} C_VEL
LIN {X 0,Y 401.291,Z 391.718,A -85,B 0,C 180,E1 -11275.409,E2 -11275.409} C_VEL
LIN {X 0,Y 399.367,Z 381.502,A -85,B 0,C 180,E1 -11277.76,E2 -11277.76} C_VEL
LIN {X 0,Y 397.124,Z 372.017,A -85,B 0,C 180,E1 -11280.084,E2 -11280.084} C_VEL
LIN {X 0,Y 397.117,Z 372.02,A -85,B 0,C 180,E1 -11283.717,E2 -11283.717} C_VEL
LIN {X 0,Y 397.095,Z 372.021,A -85,B 0,C 180,E1 -11287.209,E2 -11287.209} C_VEL
LIN {X 0,Y 397.099,Z 372.017,A -85,B 0,C 180,E1 -11290.445,E2 -11290.445} C_VEL
LIN {X 0,Y 397.098,Z 372.019,A -85,B 0,C 180,E1 -11293.648,E2 -11293.648} C_VEL
LIN {X 0,Y 397.157,Z 372.008,A -85,B 0,C 180,E1 -11296.511,E2 -11296.511} C_VEL
LIN {X 0,Y 397.118,Z 372.017,A -85,B 0,C 180,E1 -11299.55,E2 -11299.55} C_VEL
LIN {X 0,Y 397.093,Z 372.016,A -85,B 0,C 180,E1 -11302.79,E2 -11302.79} C_VEL
LIN {X 0,Y 397.112,Z 372.016,A -85,B 0,C 180,E1 -11306.282,E2 -11306.282} C_VEL
LIN {X 0,Y 397.107,Z 372.016,A -85,B 0,C 180,E1 -11310.133,E2 -11310.133} C_VEL
LIN {X 0,Y 397.188,Z 372.006,A -85,B 0,C 180,E1 -11312.609,E2 -11312.609} C_VEL
LIN {X 0,Y 397.126,Z 372.005,A -85,B 0,C 180,E1 -11315.981,E2 -11315.981} C_VEL
LIN {X 0,Y 397.131,Z 372.013,A -85,B 0,C 180,E1 -11319.704,E2 -11319.704} C_VEL
LIN {X 0,Y 397.174,Z 372.011,A -85,B 0,C 180,E1 -11322.845,E2 -11322.845} C_VEL
LIN {X 0,Y 397.218,Z 372.004,A -85,B 0,C 180,E1 -11326.679,E2 -11326.679} C_VEL
LIN {X 0,Y 397.222,Z 371.999,A -85,B 0,C 180,E1 -11329.809,E2 -11329.809} C_VEL
LIN {X 0,Y 397.356,Z 371.989,A -85,B 0,C 180,E1 -11332.888,E2 -11332.888} C_VEL
LIN {X 0,Y 397.249,Z 371.998,A -85,B 0,C 180,E1 -11334.925,E2 -11334.925} C_VEL
LIN {X 0,Y 397.444,Z 371.972,A -85,B 0,C 180,E1 -11337.973,E2 -11337.973} C_VEL
LIN {X 0,Y 397.574,Z 371.957,A -85,B 0,C 180,E1 -11340,E2 -11340} C_VEL
LIN {X 0,Y 397.375,Z 371.981,A -85,B 0,C 180,E1 -11343.042,E2 -11343.042} C_VEL
LIN {X 0,Y 397.341,Z 371.985,A -85,B 0,C 180,E1 -11346.664,E2 -11346.664} C_VEL
LIN {X 0,Y 397.245,Z 372.001,A -85,B 0,C 180,E1 -11349.162,E2 -11349.162} C_VEL
LIN {X 0,Y 397.212,Z 372.004,A -85,B 0,C 180,E1 -11352.259,E2 -11352.259} C_VEL
LIN {X 0,Y 397.172,Z 372.009,A -85,B 0,C 180,E1 -11355.393,E2 -11355.393} C_VEL
LIN {X 0,Y 397.155,Z 372.016,A -85,B 0,C 180,E1 -11358.574,E2 -11358.574} C_VEL
LIN {X 0,Y 397.09,Z 372.017,A -85,B 0,C 180,E1 -11361.819,E2 -11361.819} C_VEL
LIN {X 0,Y 397.151,Z 372.003,A -85,B 0,C 180,E1 -11365.132,E2 -11365.132} C_VEL
LIN {X 0,Y 397.156,Z 372.002,A -85,B 0,C 180,E1 -11367.777,E2 -11367.777} C_VEL
LIN {X 0,Y 397.073,Z 372.019,A -85,B 0,C 180,E1 -11370.883,E2 -11370.883} C_VEL
LIN {X 0,Y 397.122,Z 372.019,A -85,B 0,C 180,E1 -11374.494,E2 -11374.494} C_VEL
LIN {X 0,Y 397.106,Z 372.022,A -85,B 0,C 180,E1 -11378.275,E2 -11378.275} C_VEL
LIN {X 0,Y 397.154,Z 372.011,A -85,B 0,C 180,E1 -11381.994,E2 -11381.994} C_VEL
LIN {X 0,Y 397.11,Z 372.022,A -85,B 0,C 180,E1 -11385.066,E2 -11385.066} C_VEL
LIN {X 0,Y 397.109,Z 372.026,A -85,B 0,C 180,E1 -11388.015,E2 -11388.015} C_VEL
LIN {X 0,Y 397.138,Z 372.017,A -85,B 0,C 180,E1 -11391.138,E2 -11391.138} C_VEL
LIN {X 0,Y 397.121,Z 372.019,A -85,B 0,C 180,E1 -11394.497,E2 -11394.497} C_VEL
LIN {X 0,Y 397.141,Z 372.145,A -85,B 0,C 180,E1 -11397.673,E2 -11397.673} C_VEL
LIN {X 0,Y 399.134,Z 381.835,A -85,B 0,C 180,E1 -11400.461,E2 -11400.461} C_VEL
LIN {X 0,Y 402.5,Z 391.533,A -85,B 0,C 180,E1 -11400.856,E2 -11400.856} C_VEL
LIN {X 0,Y 405.091,Z 402.533,A -85,B 0,C 180,E1 -11401.22,E2 -11401.22} C_VEL
LIN {X 0,Y 403.711,Z 488.464,A -85,B 0,C 180,E1 -11402.786,E2 -11402.786} C_VEL
LIN {X 0,Y 403.278,Z 500.866,A -85,B 0,C 180,E1 -11403.197,E2 -11403.197} C_VEL
LIN {X 0,Y 402.613,Z 514.031,A -85,B 0,C 180,E1 -11403.848,E2 -11403.848} C_VEL
LIN {X 0,Y 401.853,Z 525.595,A -85,B 0,C 180,E1 -11404.63,E2 -11404.63} C_VEL
LIN {X 0,Y 401.172,Z 535.803,A -85,B 0,C 180,E1 -11405.517,E2 -11405.517} C_VEL
LIN {X 0,Y 400.117,Z 546.947,A -85,B 0,C 180,E1 -11406.722,E2 -11406.722} C_VEL
LIN {X 0,Y 399.204,Z 556.633,A -85,B 0,C 180,E1 -11408.031,E2 -11408.031} C_VEL
LIN {X 0,Y 398.237,Z 565.867,A -85,B 0,C 180,E1 -11409.602,E2 -11409.602} C_VEL
LIN {X 0,Y 397.45,Z 573.256,A -85,B 0,C 180,E1 -11411.174,E2 -11411.174} C_VEL
LIN {X 0,Y 397.016,Z 578.213,A -85,B 0,C 180,E1 -11412.487,E2 -11412.487} C_VEL
LIN {X 0,Y 396.552,Z 582.989,A -85,B 0,C 180,E1 -11414.056,E2 -11414.056} C_VEL
LIN {X 0,Y 396.221,Z 586.608,A -85,B 0,C 180,E1 -11415.622,E2 -11415.622} C_VEL
LIN {X 0,Y 396.008,Z 589.539,A -85,B 0,C 180,E1 -11417.449,E2 -11417.449} C_VEL
LIN {X 0,Y 395.86,Z 590.782,A -85,B 0,C 180,E1 -11418.739,E2 -11418.739} C_VEL
LIN {X 0,Y 395.753,Z 591.356,A -85,B 0,C 180,E1 -11419.771,E2 -11419.771} C_VEL
LIN {X 0,Y 395.755,Z 591.508,A -85,B 0,C 180,E1 -11420.803,E2 -11420.803} C_VEL
LIN {X 0,Y 395.865,Z 590.588,A -85,B 0,C 180,E1 -11422.861,E2 -11422.861} C_VEL
LIN {X 0,Y 395.913,Z 589.553,A -85,B 0,C 180,E1 -11423.886,E2 -11423.886} C_VEL
LIN {X 0,Y 395.972,Z 588.086,A -85,B 0,C 180,E1 -11424.909,E2 -11424.909} C_VEL
LIN {X 0,Y 396.153,Z 585.095,A -85,B 0,C 180,E1 -11426.44,E2 -11426.44} C_VEL
LIN {X 0,Y 396.357,Z 581.071,A -85,B 0,C 180,E1 -11427.968,E2 -11427.968} C_VEL
LIN {X 0,Y 396.73,Z 574.896,A -85,B 0,C 180,E1 -11429.746,E2 -11429.746} C_VEL
LIN {X 0,Y 397.333,Z 568.168,A -85,B 0,C 180,E1 -11431.267,E2 -11431.267} C_VEL
LIN {X 0,Y 397.978,Z 559.82,A -85,B 0,C 180,E1 -11432.783,E2 -11432.783} C_VEL
LIN {X 0,Y 398.576,Z 551.241,A -85,B 0,C 180,E1 -11434.044,E2 -11434.044} C_VEL
LIN {X 0,Y 399.147,Z 543.453,A -85,B 0,C 180,E1 -11435,E2 -11435} C_VEL
LIN {X 0,Y 398.815,Z 538.818,A -85,B 0,C 180,E1 -11435.522,E2 -11435.522} C_VEL
LIN {X 0,Y 396.611,Z 531.04,A -85,B 0,C 180,E1 -11436.355,E2 -11436.355} C_VEL
LIN {X 0,Y 394.379,Z 522.904,A -85,B 0,C 180,E1 -11437.108,E2 -11437.108} C_VEL
LIN {X 0,Y 393.968,Z 517.648,A -85,B 0,C 180,E1 -11437.494,E2 -11437.494} C_VEL
LIN {X 0,Y 394.478,Z 505.169,A -85,B 0,C 180,E1 -11438.194,E2 -11438.194} C_VEL
LIN {X 0,Y 394.904,Z 493.013,A -85,B 0,C 180,E1 -11438.668,E2 -11438.668} C_VEL
LIN {X 0,Y 395.237,Z 479.355,A -85,B 0,C 180,E1 -11438.983,E2 -11438.983} C_VEL
LIN {X 0,Y 396.179,Z 402.1,A -85,B 0,C 180,E1 -11440.38,E2 -11440.38} C_VEL
LIN {X 0,Y 392.605,Z 384.976,A -85,B 0,C 180,E1 -11440.862,E2 -11440.862} C_VEL
LIN {X 0,Y 391.693,Z 381.745,A -85,B 0,C 180,E1 -11440.973,E2 -11440.973} C_VEL
LIN {X 0,Y 390.187,Z 372.883,A -85,B 0,C 180,E1 -11443.385,E2 -11443.385} C_VEL
LIN {X 0,Y 390.146,Z 372.887,A -85,B 0,C 180,E1 -11446.751,E2 -11446.751} C_VEL
LIN {X 0,Y 390.096,Z 372.895,A -85,B 0,C 180,E1 -11450.472,E2 -11450.472} C_VEL
LIN {X 0,Y 390.093,Z 372.89,A -85,B 0,C 180,E1 -11453.35,E2 -11453.35} C_VEL
LIN {X 0,Y 390.116,Z 372.89,A -85,B 0,C 180,E1 -11456.767,E2 -11456.767} C_VEL
LIN {X 0,Y 390.046,Z 372.902,A -85,B 0,C 180,E1 -11460.298,E2 -11460.298} C_VEL
LIN {X 0,Y 390.069,Z 372.896,A -85,B 0,C 180,E1 -11464.024,E2 -11464.024} C_VEL
LIN {X 0,Y 390.046,Z 372.896,A -85,B 0,C 180,E1 -11467.55,E2 -11467.55} C_VEL
LIN {X 0,Y 390.055,Z 372.897,A -85,B 0,C 180,E1 -11470.82,E2 -11470.82} C_VEL
LIN {X 0,Y 390.057,Z 372.897,A -85,B 0,C 180,E1 -11473.886,E2 -11473.886} C_VEL
LIN {X 0,Y 390.115,Z 372.89,A -85,B 0,C 180,E1 -11476.797,E2 -11476.797} C_VEL
LIN {X 0,Y 390.075,Z 372.893,A -85,B 0,C 180,E1 -11479.562,E2 -11479.562} C_VEL
LIN {X 0,Y 390.044,Z 372.901,A -85,B 0,C 180,E1 -11482.447,E2 -11482.447} C_VEL
LIN {X 0,Y 390.064,Z 372.899,A -85,B 0,C 180,E1 -11486.044,E2 -11486.044} C_VEL
LIN {X 0,Y 390.042,Z 372.9,A -85,B 0,C 180,E1 -11489.868,E2 -11489.868} C_VEL
LIN {X 0,Y 390.108,Z 372.889,A -85,B 0,C 180,E1 -11493.231,E2 -11493.231} C_VEL
LIN {X 0,Y 390.101,Z 372.892,A -85,B 0,C 180,E1 -11496.749,E2 -11496.749} C_VEL
LIN {X 0,Y 390.114,Z 372.893,A -85,B 0,C 180,E1 -11499.983,E2 -11499.983} C_VEL
LIN {X 0,Y 390.131,Z 372.886,A -85,B 0,C 180,E1 -11503.248,E2 -11503.248} C_VEL
LIN {X 0,Y 390.187,Z 372.882,A -85,B 0,C 180,E1 -11506.561,E2 -11506.561} C_VEL
LIN {X 0,Y 390.172,Z 372.883,A -85,B 0,C 180,E1 -11509.623,E2 -11509.623} C_VEL
LIN {X 0,Y 390.31,Z 372.865,A -85,B 0,C 180,E1 -11512.759,E2 -11512.759} C_VEL
LIN {X 0,Y 390.22,Z 372.876,A -85,B 0,C 180,E1 -11514.833,E2 -11514.833} C_VEL
LIN {X 0,Y 390.413,Z 372.855,A -85,B 0,C 180,E1 -11517.936,E2 -11517.936} C_VEL
LIN {X 0,Y 390.544,Z 372.839,A -85,B 0,C 180,E1 -11520,E2 -11520} C_VEL
LIN {X 0,Y 390.31,Z 372.864,A -85,B 0,C 180,E1 -11523.096,E2 -11523.096} C_VEL
LIN {X 0,Y 390.323,Z 372.867,A -85,B 0,C 180,E1 -11526.202,E2 -11526.202} C_VEL
LIN {X 0,Y 390.307,Z 372.869,A -85,B 0,C 180,E1 -11528.282,E2 -11528.282} C_VEL
LIN {X 0,Y 390.171,Z 372.883,A -85,B 0,C 180,E1 -11532.483,E2 -11532.483} C_VEL
LIN {X 0,Y 390.132,Z 372.889,A -85,B 0,C 180,E1 -11535.677,E2 -11535.677} C_VEL
LIN {X 0,Y 390.109,Z 372.889,A -85,B 0,C 180,E1 -11538.922,E2 -11538.922} C_VEL
LIN {X 0,Y 390.048,Z 372.901,A -85,B 0,C 180,E1 -11542.233,E2 -11542.233} C_VEL
LIN {X 0,Y 390.112,Z 372.892,A -85,B 0,C 180,E1 -11545.744,E2 -11545.744} C_VEL
LIN {X 0,Y 390.051,Z 372.896,A -85,B 0,C 180,E1 -11549.11,E2 -11549.11} C_VEL
LIN {X 0,Y 390.036,Z 372.898,A -85,B 0,C 180,E1 -11552.722,E2 -11552.722} C_VEL
LIN {X 0,Y 390.052,Z 372.9,A -85,B 0,C 180,E1 -11555.826,E2 -11555.826} C_VEL
LIN {X 0,Y 390.069,Z 372.894,A -85,B 0,C 180,E1 -11559.22,E2 -11559.22} C_VEL
LIN {X 0,Y 390.118,Z 372.889,A -85,B 0,C 180,E1 -11562.388,E2 -11562.388} C_VEL
LIN {X 0,Y 390.058,Z 372.896,A -85,B 0,C 180,E1 -11565.358,E2 -11565.358} C_VEL
LIN {X 0,Y 390.027,Z 372.902,A -85,B 0,C 180,E1 -11568.187,E2 -11568.187} C_VEL
LIN {X 0,Y 390.088,Z 372.891,A -85,B 0,C 180,E1 -11570.908,E2 -11570.908} C_VEL
LIN {X 0,Y 390.084,Z 372.891,A -85,B 0,C 180,E1 -11574.794,E2 -11574.794} C_VEL
LIN {X 0,Y 390.048,Z 372.896,A -85,B 0,C 180,E1 -11578.499,E2 -11578.499} C_VEL
LIN {X 0,Y 390.143,Z 372.956,A -85,B 0,C 180,E1 -11581.087,E2 -11581.087} C_VEL
LIN {X 0,Y 392.759,Z 386.022,A -85,B 0,C 180,E1 -11584.024,E2 -11584.024} C_VEL
LIN {X 0,Y 393.363,Z 391.371,A -85,B 0,C 180,E1 -11585.175,E2 -11585.175} C_VEL
LIN {X 0,Y 391.956,Z 409.275,A -85,B 0,C 180,E1 -11588.811,E2 -11588.811} C_VEL
LIN {X 0,Y 391.572,Z 415.301,A -85,B 0,C 180,E1 -11590.028,E2 -11590.028} C_VEL
LIN {X 0,Y 395.879,Z 447.519,A -85,B 0,C 180,E1 -11590.818,E2 -11590.818} C_VEL
LIN {X 0,Y 394.879,Z 524.06,A -85,B 0,C 180,E1 -11592.222,E2 -11592.222} C_VEL
LIN {X 0,Y 394.327,Z 537.323,A -85,B 0,C 180,E1 -11592.664,E2 -11592.664} C_VEL
LIN {X 0,Y 393.641,Z 549.505,A -85,B 0,C 180,E1 -11593.269,E2 -11593.269} C_VEL
LIN {X 0,Y 392.877,Z 560.987,A -85,B 0,C 180,E1 -11594.036,E2 -11594.036} C_VEL
LIN {X 0,Y 391.982,Z 572.782,A -85,B 0,C 180,E1 -11595.065,E2 -11595.065} C_VEL
LIN {X 0,Y 391.365,Z 581.748,A -85,B 0,C 180,E1 -11596.035,E2 -11596.035} C_VEL
LIN {X 0,Y 390.61,Z 591.137,A -85,B 0,C 180,E1 -11597.267,E2 -11597.267} C_VEL
LIN {X 0,Y 390.026,Z 599.266,A -85,B 0,C 180,E1 -11598.568,E2 -11598.568} C_VEL
LIN {X 0,Y 389.416,Z 607.227,A -85,B 0,C 180,E1 -11600.128,E2 -11600.128} C_VEL
LIN {X 0,Y 389.073,Z 613.581,A -85,B 0,C 180,E1 -11601.691,E2 -11601.691} C_VEL
LIN {X 0,Y 388.823,Z 618.629,A -85,B 0,C 180,E1 -11603.253,E2 -11603.253} C_VEL
LIN {X 0,Y 388.775,Z 622.531,A -85,B 0,C 180,E1 -11604.814,E2 -11604.814} C_VEL
LIN {X 0,Y 388.72,Z 624.535,A -85,B 0,C 180,E1 -11605.853,E2 -11605.853} C_VEL
LIN {X 0,Y 388.71,Z 626.12,A -85,B 0,C 180,E1 -11606.891,E2 -11606.891} C_VEL
LIN {X 0,Y 388.793,Z 627.283,A -85,B 0,C 180,E1 -11607.928,E2 -11607.928} C_VEL
LIN {X 0,Y 388.76,Z 628,A -85,B 0,C 180,E1 -11608.964,E2 -11608.964} C_VEL
LIN {X 0,Y 388.759,Z 628.271,A -85,B 0,C 180,E1 -11611.036,E2 -11611.036} C_VEL
LIN {X 0,Y 388.754,Z 627.813,A -85,B 0,C 180,E1 -11612.072,E2 -11612.072} C_VEL
LIN {X 0,Y 388.707,Z 625.63,A -85,B 0,C 180,E1 -11614.147,E2 -11614.147} C_VEL
LIN {X 0,Y 388.744,Z 623.939,A -85,B 0,C 180,E1 -11615.186,E2 -11615.186} C_VEL
LIN {X 0,Y 388.842,Z 620.549,A -85,B 0,C 180,E1 -11616.747,E2 -11616.747} C_VEL
LIN {X 0,Y 389.113,Z 616.097,A -85,B 0,C 180,E1 -11618.308,E2 -11618.308} C_VEL
LIN {X 0,Y 389.609,Z 609.388,A -85,B 0,C 180,E1 -11620.129,E2 -11620.129} C_VEL
LIN {X 0,Y 390.291,Z 602.084,A -85,B 0,C 180,E1 -11621.688,E2 -11621.688} C_VEL
LIN {X 0,Y 391.28,Z 593.049,A -85,B 0,C 180,E1 -11623.238,E2 -11623.238} C_VEL
LIN {X 0,Y 392.099,Z 583.548,A -85,B 0,C 180,E1 -11624.557,E2 -11624.557} C_VEL
LIN {X 0,Y 393.091,Z 573.417,A -85,B 0,C 180,E1 -11625.689,E2 -11625.689} C_VEL
LIN {X 0,Y 394.176,Z 561.986,A -85,B 0,C 180,E1 -11626.708,E2 -11626.708} C_VEL
LIN {X 0,Y 395.182,Z 550.061,A -85,B 0,C 180,E1 -11627.53,E2 -11627.53} C_VEL
LIN {X 0,Y 396.097,Z 536.834,A -85,B 0,C 180,E1 -11628.189,E2 -11628.189} C_VEL
LIN {X 0,Y 396.695,Z 523.826,A -85,B 0,C 180,E1 -11628.625,E2 -11628.625} C_VEL
LIN {X 0,Y 397.824,Z 446.33,A -85,B 0,C 180,E1 -11630.071,E2 -11630.071} C_VEL
LIN {X 0,Y 394.347,Z 424.529,A -85,B 0,C 180,E1 -11630.703,E2 -11630.703} C_VEL
LIN {X 0,Y 392.492,Z 414.84,A -85,B 0,C 180,E1 -11631.022,E2 -11631.022} C_VEL
LIN {X 0,Y 393.764,Z 400.757,A -85,B 0,C 180,E1 -11633.956,E2 -11633.956} C_VEL
LIN {X 0,Y 394.449,Z 394.269,A -85,B 0,C 180,E1 -11635.316,E2 -11635.316} C_VEL
LIN {X 0,Y 393.514,Z 388.025,A -85,B 0,C 180,E1 -11636.75,E2 -11636.75} C_VEL
LIN {X 0,Y 391.172,Z 377.432,A -85,B 0,C 180,E1 -11639.313,E2 -11639.313} C_VEL
LIN {X 0,Y 390.058,Z 372.895,A -85,B 0,C 180,E1 -11640.484,E2 -11640.484} C_VEL
LIN {X 0,Y 390.066,Z 372.899,A -85,B 0,C 180,E1 -11644.024,E2 -11644.024} C_VEL
LIN {X 0,Y 390.043,Z 372.901,A -85,B 0,C 180,E1 -11647.551,E2 -11647.551} C_VEL
LIN {X 0,Y 390.053,Z 372.894,A -85,B 0,C 180,E1 -11650.821,E2 -11650.821} C_VEL
LIN {X 0,Y 390.055,Z 372.896,A -85,B 0,C 180,E1 -11653.886,E2 -11653.886} C_VEL
LIN {X 0,Y 390.111,Z 372.885,A -85,B 0,C 180,E1 -11656.797,E2 -11656.797} C_VEL
LIN {X 0,Y 390.072,Z 372.894,A -85,B 0,C 180,E1 -11659.563,E2 -11659.563} C_VEL
LIN {X 0,Y 390.041,Z 372.894,A -85,B 0,C 180,E1 -11662.448,E2 -11662.448} C_VEL
LIN {X 0,Y 390.062,Z 372.896,A -85,B 0,C 180,E1 -11666.045,E2 -11666.045} C_VEL
LIN {X 0,Y 390.045,Z 372.897,A -85,B 0,C 180,E1 -11669.867,E2 -11669.867} C_VEL
LIN {X 0,Y 390.107,Z 372.885,A -85,B 0,C 180,E1 -11673.231,E2 -11673.231} C_VEL
LIN {X 0,Y 390.099,Z 372.882,A -85,B 0,C 180,E1 -11676.75,E2 -11676.75} C_VEL
LIN {X 0,Y 390.096,Z 372.888,A -85,B 0,C 180,E1 -11679.983,E2 -11679.983} C_VEL
LIN {X 0,Y 390.13,Z 372.89,A -85,B 0,C 180,E1 -11683.248,E2 -11683.248} C_VEL
LIN {X 0,Y 390.186,Z 372.879,A -85,B 0,C 180,E1 -11686.561,E2 -11686.561} C_VEL
LIN {X 0,Y 390.171,Z 372.878,A -85,B 0,C 180,E1 -11689.623,E2 -11689.623} C_VEL
LIN {X 0,Y 390.31,Z 372.868,A -85,B 0,C 180,E1 -11692.759,E2 -11692.759} C_VEL
LIN {X 0,Y 390.22,Z 372.873,A -85,B 0,C 180,E1 -11694.834,E2 -11694.834} C_VEL
LIN {X 0,Y 390.413,Z 372.848,A -85,B 0,C 180,E1 -11697.937,E2 -11697.937} C_VEL
LIN {X 0,Y 390.544,Z 372.832,A -85,B 0,C 180,E1 -11700,E2 -11700} C_VEL
LIN {X 0,Y 390.309,Z 372.86,A -85,B 0,C 180,E1 -11703.097,E2 -11703.097} C_VEL
LIN {X 0,Y 390.295,Z 372.863,A -85,B 0,C 180,E1 -11706.66,E2 -11706.66} C_VEL
LIN {X 0,Y 390.198,Z 372.878,A -85,B 0,C 180,E1 -11709.329,E2 -11709.329} C_VEL
LIN {X 0,Y 390.187,Z 372.877,A -85,B 0,C 180,E1 -11713.439,E2 -11713.439} C_VEL
LIN {X 0,Y 390.142,Z 372.882,A -85,B 0,C 180,E1 -11717.308,E2 -11717.308} C_VEL
LIN {X 0,Y 390.081,Z 372.892,A -85,B 0,C 180,E1 -11720.471,E2 -11720.471} C_VEL
LIN {X 0,Y 390.083,Z 372.892,A -85,B 0,C 180,E1 -11723.352,E2 -11723.352} C_VEL
LIN {X 0,Y 390.108,Z 372.876,A -85,B 0,C 180,E1 -11726.769,E2 -11726.769} C_VEL
LIN {X 0,Y 390.034,Z 372.901,A -85,B 0,C 180,E1 -11730.301,E2 -11730.301} C_VEL
LIN {X 0,Y 390.064,Z 372.897,A -85,B 0,C 180,E1 -11734.026,E2 -11734.026} C_VEL
LIN {X 0,Y 390.043,Z 372.899,A -85,B 0,C 180,E1 -11737.552,E2 -11737.552} C_VEL
LIN {X 0,Y 390.08,Z 372.896,A -85,B 0,C 180,E1 -11740.827,E2 -11740.827} C_VEL
LIN {X 0,Y 390.102,Z 372.896,A -85,B 0,C 180,E1 -11743.895,E2 -11743.895} C_VEL
LIN {X 0,Y 390.079,Z 372.9,A -85,B 0,C 180,E1 -11747.621,E2 -11747.621} C_VEL
LIN {X 0,Y 390.095,Z 372.894,A -85,B 0,C 180,E1 -11750.909,E2 -11750.909} C_VEL
LIN {X 0,Y 390.087,Z 372.895,A -85,B 0,C 180,E1 -11754.794,E2 -11754.794} C_VEL
LIN {X 0,Y 390.081,Z 372.913,A -85,B 0,C 180,E1 -11757.283,E2 -11757.283} C_VEL
LIN {X 0,Y 392.05,Z 382.141,A -85,B 0,C 180,E1 -11759.999,E2 -11759.999} C_VEL
LIN {X 0,Y 396.11,Z 393.341,A -85,B 0,C 180,E1 -11760.494,E2 -11760.494} C_VEL
LIN {X 0,Y 398.502,Z 403.527,A -85,B 0,C 180,E1 -11760.84,E2 -11760.84} C_VEL
LIN {X 0,Y 397.095,Z 489.02,A -85,B 0,C 180,E1 -11762.428,E2 -11762.428} C_VEL
LIN {X 0,Y 396.633,Z 501.548,A -85,B 0,C 180,E1 -11762.854,E2 -11762.854} C_VEL
LIN {X 0,Y 395.93,Z 514.618,A -85,B 0,C 180,E1 -11763.514,E2 -11763.514} C_VEL
LIN {X 0,Y 395.134,Z 526.104,A -85,B 0,C 180,E1 -11764.308,E2 -11764.308} C_VEL
LIN {X 0,Y 394.231,Z 538.119,A -85,B 0,C 180,E1 -11765.394,E2 -11765.394} C_VEL
LIN {X 0,Y 393.196,Z 548.486,A -85,B 0,C 180,E1 -11766.566,E2 -11766.566} C_VEL
LIN {X 0,Y 392.274,Z 557.89,A -85,B 0,C 180,E1 -11767.9,E2 -11767.9} C_VEL
LIN {X 0,Y 391.257,Z 566.999,A -85,B 0,C 180,E1 -11769.504,E2 -11769.504} C_VEL
LIN {X 0,Y 390.443,Z 574.196,A -85,B 0,C 180,E1 -11771.095,E2 -11771.095} C_VEL
LIN {X 0,Y 389.858,Z 580.315,A -85,B 0,C 180,E1 -11772.832,E2 -11772.832} C_VEL
LIN {X 0,Y 389.299,Z 585.612,A -85,B 0,C 180,E1 -11774.825,E2 -11774.825} C_VEL
LIN {X 0,Y 389,Z 588.6,A -85,B 0,C 180,E1 -11776.416,E2 -11776.416} C_VEL
LIN {X 0,Y 388.927,Z 590.026,A -85,B 0,C 180,E1 -11777.477,E2 -11777.477} C_VEL
LIN {X 0,Y 388.687,Z 591.636,A -85,B 0,C 180,E1 -11779.583,E2 -11779.583} C_VEL
LIN {X 0,Y 388.665,Z 591.852,A -85,B 0,C 180,E1 -11780.634,E2 -11780.634} C_VEL
LIN {X 0,Y 388.685,Z 591.631,A -85,B 0,C 180,E1 -11781.683,E2 -11781.683} C_VEL
LIN {X 0,Y 388.774,Z 591.014,A -85,B 0,C 180,E1 -11782.73,E2 -11782.73} C_VEL
LIN {X 0,Y 388.837,Z 590.014,A -85,B 0,C 180,E1 -11783.774,E2 -11783.774} C_VEL
LIN {X 0,Y 388.877,Z 588.618,A -85,B 0,C 180,E1 -11784.816,E2 -11784.816} C_VEL
LIN {X 0,Y 389.049,Z 585.695,A -85,B 0,C 180,E1 -11786.375,E2 -11786.375} C_VEL
LIN {X 0,Y 389.295,Z 581.747,A -85,B 0,C 180,E1 -11787.931,E2 -11787.931} C_VEL
LIN {X 0,Y 389.575,Z 576.675,A -85,B 0,C 180,E1 -11789.483,E2 -11789.483} C_VEL
LIN {X 0,Y 390.138,Z 570.276,A -85,B 0,C 180,E1 -11791.032,E2 -11791.032} C_VEL
LIN {X 0,Y 390.777,Z 562.325,A -85,B 0,C 180,E1 -11792.577,E2 -11792.577} C_VEL
LIN {X 0,Y 391.425,Z 554.224,A -85,B 0,C 180,E1 -11793.861,E2 -11793.861} C_VEL
LIN {X 0,Y 392.172,Z 544.355,A -85,B 0,C 180,E1 -11795.141,E2 -11795.141} C_VEL
LIN {X 0,Y 393.026,Z 533.185,A -85,B 0,C 180,E1 -11796.288,E2 -11796.288} C_VEL
LIN {X 0,Y 393.774,Z 522.254,A -85,B 0,C 180,E1 -11797.177,E2 -11797.177} C_VEL
LIN {X 0,Y 393.968,Z 517.648,A -85,B 0,C 180,E1 -11797.494,E2 -11797.494} C_VEL
LIN {X 0,Y 393.571,Z 512.271,A -85,B 0,C 180,E1 -11797.85,E2 -11797.85} C_VEL
LIN {X 0,Y 391.167,Z 503.437,A -85,B 0,C 180,E1 -11798.41,E2 -11798.41} C_VEL
LIN {X 0,Y 388.717,Z 494.387,A -85,B 0,C 180,E1 -11798.875,E2 -11798.875} C_VEL
LIN {X 0,Y 388.187,Z 488.677,A -85,B 0,C 180,E1 -11799.072,E2 -11799.072} C_VEL
LIN {X 0,Y 389.404,Z 403.078,A -85,B 0,C 180,E1 -11800.666,E2 -11800.666} C_VEL
LIN {X 0,Y 385.97,Z 386.79,A -85,B 0,C 180,E1 -11801.137,E2 -11801.137} C_VEL
LIN {X 0,Y 384.601,Z 382.037,A -85,B 0,C 180,E1 -11801.306,E2 -11801.306} C_VEL
LIN {X 0,Y 383.141,Z 373.761,A -85,B 0,C 180,E1 -11803.632,E2 -11803.632} C_VEL
LIN {X 0,Y 383.1,Z 373.761,A -85,B 0,C 180,E1 -11807.455,E2 -11807.455} C_VEL
LIN {X 0,Y 383.038,Z 373.773,A -85,B 0,C 180,E1 -11810.649,E2 -11810.649} C_VEL
LIN {X 0,Y 383.037,Z 373.77,A -85,B 0,C 180,E1 -11813.806,E2 -11813.806} C_VEL
LIN {X 0,Y 383.059,Z 373.766,A -85,B 0,C 180,E1 -11817.301,E2 -11817.301} C_VEL
LIN {X 0,Y 382.988,Z 373.777,A -85,B 0,C 180,E1 -11820.917,E2 -11820.917} C_VEL
LIN {X 0,Y 383.019,Z 373.775,A -85,B 0,C 180,E1 -11824.667,E2 -11824.667} C_VEL
LIN {X 0,Y 383.001,Z 373.776,A -85,B 0,C 180,E1 -11827.903,E2 -11827.903} C_VEL
LIN {X 0,Y 382.982,Z 373.776,A -85,B 0,C 180,E1 -11831.346,E2 -11831.346} C_VEL
LIN {X 0,Y 383.006,Z 373.778,A -85,B 0,C 180,E1 -11834.304,E2 -11834.304} C_VEL
LIN {X 0,Y 383.073,Z 373.765,A -85,B 0,C 180,E1 -11837.248,E2 -11837.248} C_VEL
LIN {X 0,Y 383.019,Z 373.776,A -85,B 0,C 180,E1 -11840.411,E2 -11840.411} C_VEL
LIN {X 0,Y 383.023,Z 373.775,A -85,B 0,C 180,E1 -11844.044,E2 -11844.044} C_VEL
LIN {X 0,Y 382.982,Z 373.777,A -85,B 0,C 180,E1 -11847.577,E2 -11847.577} C_VEL
LIN {X 0,Y 382.987,Z 373.78,A -85,B 0,C 180,E1 -11850.299,E2 -11850.299} C_VEL
LIN {X 0,Y 383.075,Z 373.769,A -85,B 0,C 180,E1 -11854.02,E2 -11854.02} C_VEL
LIN {X 0,Y 383.011,Z 373.773,A -85,B 0,C 180,E1 -11857.335,E2 -11857.335} C_VEL
LIN {X 0,Y 383.066,Z 373.768,A -85,B 0,C 180,E1 -11860.716,E2 -11860.716} C_VEL
LIN {X 0,Y 383.075,Z 373.77,A -85,B 0,C 180,E1 -11864.026,E2 -11864.026} C_VEL
LIN {X 0,Y 383.135,Z 373.758,A -85,B 0,C 180,E1 -11867.284,E2 -11867.284} C_VEL
LIN {X 0,Y 383.149,Z 373.759,A -85,B 0,C 180,E1 -11870.498,E2 -11870.498} C_VEL
LIN {X 0,Y 383.265,Z 373.743,A -85,B 0,C 180,E1 -11872.625,E2 -11872.625} C_VEL
LIN {X 0,Y 383.192,Z 373.751,A -85,B 0,C 180,E1 -11874.738,E2 -11874.738} C_VEL
LIN {X 0,Y 383.38,Z 373.731,A -85,B 0,C 180,E1 -11877.899,E2 -11877.899} C_VEL
LIN {X 0,Y 383.513,Z 373.715,A -85,B 0,C 180,E1 -11880,E2 -11880} C_VEL
LIN {X 0,Y 383.246,Z 373.744,A -85,B 0,C 180,E1 -11883.153,E2 -11883.153} C_VEL
LIN {X 0,Y 383.28,Z 373.744,A -85,B 0,C 180,E1 -11886.316,E2 -11886.316} C_VEL
LIN {X 0,Y 383.253,Z 373.746,A -85,B 0,C 180,E1 -11888.436,E2 -11888.436} C_VEL
LIN {X 0,Y 383.101,Z 373.764,A -85,B 0,C 180,E1 -11891.642,E2 -11891.642} C_VEL
LIN {X 0,Y 383.105,Z 373.761,A -85,B 0,C 180,E1 -11894.882,E2 -11894.882} C_VEL
LIN {X 0,Y 383.086,Z 373.769,A -85,B 0,C 180,E1 -11898.172,E2 -11898.172} C_VEL
LIN {X 0,Y 383.003,Z 373.776,A -85,B 0,C 180,E1 -11901.53,E2 -11901.53} C_VEL
LIN {X 0,Y 383.045,Z 373.768,A -85,B 0,C 180,E1 -11904.961,E2 -11904.961} C_VEL
LIN {X 0,Y 383.01,Z 373.774,A -85,B 0,C 180,E1 -11908.495,E2 -11908.495} C_VEL
LIN {X 0,Y 383.003,Z 373.778,A -85,B 0,C 180,E1 -11912.15,E2 -11912.15} C_VEL
LIN {X 0,Y 383.012,Z 373.773,A -85,B 0,C 180,E1 -11914.668,E2 -11914.668} C_VEL
LIN {X 0,Y 382.998,Z 373.779,A -85,B 0,C 180,E1 -11917.905,E2 -11917.905} C_VEL
LIN {X 0,Y 383.042,Z 373.77,A -85,B 0,C 180,E1 -11921.34,E2 -11921.34} C_VEL
LIN {X 0,Y 383.032,Z 373.772,A -85,B 0,C 180,E1 -11924.31,E2 -11924.31} C_VEL
LIN {X 0,Y 383.006,Z 373.774,A -85,B 0,C 180,E1 -11927.241,E2 -11927.241} C_VEL
LIN {X 0,Y 383.012,Z 373.773,A -85,B 0,C 180,E1 -11930.414,E2 -11930.414} C_VEL
LIN {X 0,Y 383.024,Z 373.775,A -85,B 0,C 180,E1 -11934.045,E2 -11934.045} C_VEL
LIN {X 0,Y 383.035,Z 373.776,A -85,B 0,C 180,E1 -11937.854,E2 -11937.854} C_VEL
LIN {X 0,Y 383.076,Z 373.86,A -85,B 0,C 180,E1 -11940.837,E2 -11940.837} C_VEL
LIN {X 0,Y 385.61,Z 386.389,A -85,B 0,C 180,E1 -11943.715,E2 -11943.715} C_VEL
LIN {X 0,Y 386.411,Z 392.137,A -85,B 0,C 180,E1 -11944.985,E2 -11944.985} C_VEL
LIN {X 0,Y 385.003,Z 409.541,A -85,B 0,C 180,E1 -11948.588,E2 -11948.588} C_VEL
LIN {X 0,Y 384.59,Z 414.968,A -85,B 0,C 180,E1 -11949.705,E2 -11949.705} C_VEL
LIN {X 0,Y 389.057,Z 447.83,A -85,B 0,C 180,E1 -11950.532,E2 -11950.532} C_VEL
LIN {X 0,Y 388.004,Z 523.133,A -85,B 0,C 180,E1 -11951.93,E2 -11951.93} C_VEL
LIN {X 0,Y 387.501,Z 536.623,A -85,B 0,C 180,E1 -11952.383,E2 -11952.383} C_VEL
LIN {X 0,Y 386.75,Z 549.47,A -85,B 0,C 180,E1 -11953.029,E2 -11953.029} C_VEL
LIN {X 0,Y 385.889,Z 561.672,A -85,B 0,C 180,E1 -11953.875,E2 -11953.875} C_VEL
LIN {X 0,Y 384.967,Z 573.275,A -85,B 0,C 180,E1 -11954.921,E2 -11954.921} C_VEL
LIN {X 0,Y 384.277,Z 583.445,A -85,B 0,C 180,E1 -11956.074,E2 -11956.074} C_VEL
LIN {X 0,Y 383.498,Z 592.277,A -85,B 0,C 180,E1 -11957.296,E2 -11957.296} C_VEL
LIN {X 0,Y 382.736,Z 601.518,A -85,B 0,C 180,E1 -11958.884,E2 -11958.884} C_VEL
LIN {X 0,Y 382.222,Z 608.956,A -85,B 0,C 180,E1 -11960.475,E2 -11960.475} C_VEL
LIN {X 0,Y 381.905,Z 614.917,A -85,B 0,C 180,E1 -11962.067,E2 -11962.067} C_VEL
LIN {X 0,Y 381.673,Z 620.217,A -85,B 0,C 180,E1 -11963.9,E2 -11963.9} C_VEL
LIN {X 0,Y 381.645,Z 624.122,A -85,B 0,C 180,E1 -11965.776,E2 -11965.776} C_VEL
LIN {X 0,Y 381.615,Z 625.722,A -85,B 0,C 180,E1 -11966.833,E2 -11966.833} C_VEL
LIN {X 0,Y 381.693,Z 626.91,A -85,B 0,C 180,E1 -11967.89,E2 -11967.89} C_VEL
LIN {X 0,Y 381.692,Z 627.646,A -85,B 0,C 180,E1 -11968.945,E2 -11968.945} C_VEL
LIN {X 0,Y 381.69,Z 627.944,A -85,B 0,C 180,E1 -11971.055,E2 -11971.055} C_VEL
LIN {X 0,Y 381.653,Z 627.507,A -85,B 0,C 180,E1 -11972.111,E2 -11972.111} C_VEL
LIN {X 0,Y 381.632,Z 625.359,A -85,B 0,C 180,E1 -11974.224,E2 -11974.224} C_VEL
LIN {X 0,Y 381.678,Z 622.07,A -85,B 0,C 180,E1 -11976.107,E2 -11976.107} C_VEL
LIN {X 0,Y 381.94,Z 617.525,A -85,B 0,C 180,E1 -11977.932,E2 -11977.932} C_VEL
LIN {X 0,Y 382.432,Z 611.32,A -85,B 0,C 180,E1 -11979.787,E2 -11979.787} C_VEL
LIN {X 0,Y 383.028,Z 604.582,A -85,B 0,C 180,E1 -11981.376,E2 -11981.376} C_VEL
LIN {X 0,Y 384.001,Z 596.251,A -85,B 0,C 180,E1 -11982.956,E2 -11982.956} C_VEL
LIN {X 0,Y 384.909,Z 586.565,A -85,B 0,C 180,E1 -11984.428,E2 -11984.428} C_VEL
LIN {X 0,Y 385.987,Z 576.022,A -85,B 0,C 180,E1 -11985.714,E2 -11985.714} C_VEL
LIN {X 0,Y 387.138,Z 565.375,A -85,B 0,C 180,E1 -11986.749,E2 -11986.749} C_VEL
LIN {X 0,Y 388.189,Z 553.476,A -85,B 0,C 180,E1 -11987.653,E2 -11987.653} C_VEL
LIN {X 0,Y 389.162,Z 541.116,A -85,B 0,C 180,E1 -11988.355,E2 -11988.355} C_VEL
LIN {X 0,Y 389.925,Z 528.397,A -85,B 0,C 180,E1 -11988.862,E2 -11988.862} C_VEL
LIN {X 0,Y 390.321,Z 513.419,A -85,B 0,C 180,E1 -11989.215,E2 -11989.215} C_VEL
LIN {X 0,Y 391.253,Z 446.866,A -85,B 0,C 180,E1 -11990.459,E2 -11990.459} C_VEL
LIN {X 0,Y 387.311,Z 422.878,A -85,B 0,C 180,E1 -11991.182,E2 -11991.182} C_VEL
LIN {X 0,Y 385.671,Z 414.475,A -85,B 0,C 180,E1 -11991.474,E2 -11991.474} C_VEL
LIN {X 0,Y 387.233,Z 398.63,A -85,B 0,C 180,E1 -11994.843,E2 -11994.843} C_VEL
LIN {X 0,Y 387.465,Z 394.219,A -85,B 0,C 180,E1 -11995.805,E2 -11995.805} C_VEL
LIN {X 0,Y 385.167,Z 382.726,A -85,B 0,C 180,E1 -11998.584,E2 -11998.584} C_VEL
LIN {X 0,Y 383.009,Z 373.772,A -85,B 0,C 180,E1 -12000.915,E2 -12000.915} C_VEL
LIN {X 0,Y 383.016,Z 373.777,A -85,B 0,C 180,E1 -12004.339,E2 -12004.339} C_VEL
LIN {X 0,Y 382.995,Z 373.778,A -85,B 0,C 180,E1 -12007.268,E2 -12007.268} C_VEL
LIN {X 0,Y 383.006,Z 373.776,A -85,B 0,C 180,E1 -12009.958,E2 -12009.958} C_VEL
LIN {X 0,Y 383.001,Z 373.772,A -85,B 0,C 180,E1 -12012.778,E2 -12012.778} C_VEL
LIN {X 0,Y 383.035,Z 373.77,A -85,B 0,C 180,E1 -12015.795,E2 -12015.795} C_VEL
LIN {X 0,Y 383.039,Z 373.766,A -85,B 0,C 180,E1 -12018.786,E2 -12018.786} C_VEL
LIN {X 0,Y 382.998,Z 373.774,A -85,B 0,C 180,E1 -12022.095,E2 -12022.095} C_VEL
LIN {X 0,Y 383.012,Z 373.775,A -85,B 0,C 180,E1 -12025.332,E2 -12025.332} C_VEL
LIN {X 0,Y 382.98,Z 373.779,A -85,B 0,C 180,E1 -12029.081,E2 -12029.081} C_VEL
LIN {X 0,Y 383.05,Z 373.768,A -85,B 0,C 180,E1 -12032.698,E2 -12032.698} C_VEL
LIN {X 0,Y 383.045,Z 373.751,A -85,B 0,C 180,E1 -12035.039,E2 -12035.039} C_VEL
LIN {X 0,Y 382.986,Z 373.776,A -85,B 0,C 180,E1 -12038.469,E2 -12038.469} C_VEL
LIN {X 0,Y 383.081,Z 373.765,A -85,B 0,C 180,E1 -12041.828,E2 -12041.828} C_VEL
LIN {X 0,Y 383.104,Z 373.76,A -85,B 0,C 180,E1 -12045.118,E2 -12045.118} C_VEL
LIN {X 0,Y 383.1,Z 373.761,A -85,B 0,C 180,E1 -12048.358,E2 -12048.358} C_VEL
LIN {X 0,Y 383.296,Z 373.738,A -85,B 0,C 180,E1 -12051.933,E2 -12051.933} C_VEL
LIN {X 0,Y 383.192,Z 373.747,A -85,B 0,C 180,E1 -12054.739,E2 -12054.739} C_VEL
LIN {X 0,Y 383.38,Z 373.724,A -85,B 0,C 180,E1 -12057.899,E2 -12057.899} C_VEL
LIN {X 0,Y 383.513,Z 373.708,A -85,B 0,C 180,E1 -12060,E2 -12060} C_VEL
LIN {X 0,Y 383.245,Z 373.74,A -85,B 0,C 180,E1 -12063.154,E2 -12063.154} C_VEL
LIN {X 0,Y 383.254,Z 373.741,A -85,B 0,C 180,E1 -12066.652,E2 -12066.652} C_VEL
LIN {X 0,Y 383.144,Z 373.756,A -85,B 0,C 180,E1 -12069.503,E2 -12069.503} C_VEL
LIN {X 0,Y 383.118,Z 373.757,A -85,B 0,C 180,E1 -12073.537,E2 -12073.537} C_VEL
LIN {X 0,Y 383.088,Z 373.76,A -85,B 0,C 180,E1 -12077.455,E2 -12077.455} C_VEL
LIN {X 0,Y 383.022,Z 373.77,A -85,B 0,C 180,E1 -12080.648,E2 -12080.648} C_VEL
LIN {X 0,Y 383.027,Z 373.772,A -85,B 0,C 180,E1 -12083.808,E2 -12083.808} C_VEL
LIN {X 0,Y 383.074,Z 373.751,A -85,B 0,C 180,E1 -12086.124,E2 -12086.124} C_VEL
LIN {X 0,Y 383.035,Z 373.77,A -85,B 0,C 180,E1 -12088.494,E2 -12088.494} C_VEL
LIN {X 0,Y 383.005,Z 373.776,A -85,B 0,C 180,E1 -12092.151,E2 -12092.151} C_VEL
LIN {X 0,Y 383.014,Z 373.775,A -85,B 0,C 180,E1 -12094.669,E2 -12094.669} C_VEL
LIN {X 0,Y 383,Z 373.779,A -85,B 0,C 180,E1 -12097.905,E2 -12097.905} C_VEL
LIN {X 0,Y 383.044,Z 373.773,A -85,B 0,C 180,E1 -12101.34,E2 -12101.34} C_VEL
LIN {X 0,Y 383.034,Z 373.779,A -85,B 0,C 180,E1 -12104.311,E2 -12104.311} C_VEL
LIN {X 0,Y 383.038,Z 373.774,A -85,B 0,C 180,E1 -12107.245,E2 -12107.245} C_VEL
LIN {X 0,Y 383.022,Z 373.777,A -85,B 0,C 180,E1 -12110.413,E2 -12110.413} C_VEL
LIN {X 0,Y 383.027,Z 373.774,A -85,B 0,C 180,E1 -12114.046,E2 -12114.046} C_VEL
LIN {X 0,Y 383.033,Z 373.803,A -85,B 0,C 180,E1 -12116.917,E2 -12116.917} C_VEL
LIN {X 0,Y 384.965,Z 382.737,A -85,B 0,C 180,E1 -12119.55,E2 -12119.55} C_VEL
LIN {X 0,Y 389.758,Z 395.173,A -85,B 0,C 180,E1 -12120.121,E2 -12120.121} C_VEL
LIN {X 0,Y 392.019,Z 404.765,A -85,B 0,C 180,E1 -12120.457,E2 -12120.457} C_VEL
LIN {X 0,Y 390.504,Z 489.259,A -85,B 0,C 180,E1 -12122.047,E2 -12122.047} C_VEL
LIN {X 0,Y 390.044,Z 501.48,A -85,B 0,C 180,E1 -12122.466,E2 -12122.466} C_VEL
LIN {X 0,Y 389.325,Z 514.07,A -85,B 0,C 180,E1 -12123.101,E2 -12123.101} C_VEL
LIN {X 0,Y 388.559,Z 524.925,A -85,B 0,C 180,E1 -12123.841,E2 -12123.841} C_VEL
LIN {X 0,Y 387.788,Z 535.436,A -85,B 0,C 180,E1 -12124.757,E2 -12124.757} C_VEL
LIN {X 0,Y 386.632,Z 546.767,A -85,B 0,C 180,E1 -12126.002,E2 -12126.002} C_VEL
LIN {X 0,Y 385.673,Z 555.693,A -85,B 0,C 180,E1 -12127.218,E2 -12127.218} C_VEL
LIN {X 0,Y 384.712,Z 564.546,A -85,B 0,C 180,E1 -12128.7,E2 -12128.7} C_VEL
LIN {X 0,Y 383.824,Z 571.779,A -85,B 0,C 180,E1 -12130.2,E2 -12130.2} C_VEL
LIN {X 0,Y 383.11,Z 578.061,A -85,B 0,C 180,E1 -12131.829,E2 -12131.829} C_VEL
LIN {X 0,Y 382.591,Z 583.013,A -85,B 0,C 180,E1 -12133.458,E2 -12133.458} C_VEL
LIN {X 0,Y 382.185,Z 586.797,A -85,B 0,C 180,E1 -12135.082,E2 -12135.082} C_VEL
LIN {X 0,Y 381.957,Z 588.735,A -85,B 0,C 180,E1 -12136.161,E2 -12136.161} C_VEL
LIN {X 0,Y 381.88,Z 590.26,A -85,B 0,C 180,E1 -12137.266,E2 -12137.266} C_VEL
LIN {X 0,Y 381.628,Z 591.917,A -85,B 0,C 180,E1 -12139.388,E2 -12139.388} C_VEL
LIN {X 0,Y 381.59,Z 592.173,A -85,B 0,C 180,E1 -12140.459,E2 -12140.459} C_VEL
LIN {X 0,Y 381.6,Z 592.02,A -85,B 0,C 180,E1 -12141.528,E2 -12141.528} C_VEL
LIN {X 0,Y 381.662,Z 591.44,A -85,B 0,C 180,E1 -12142.594,E2 -12142.594} C_VEL
LIN {X 0,Y 381.755,Z 590.332,A -85,B 0,C 180,E1 -12143.791,E2 -12143.791} C_VEL
LIN {X 0,Y 381.824,Z 587.335,A -85,B 0,C 180,E1 -12145.778,E2 -12145.778} C_VEL
LIN {X 0,Y 382.123,Z 583.814,A -85,B 0,C 180,E1 -12147.365,E2 -12147.365} C_VEL
LIN {X 0,Y 382.311,Z 579.22,A -85,B 0,C 180,E1 -12148.947,E2 -12148.947} C_VEL
LIN {X 0,Y 382.988,Z 572.262,A -85,B 0,C 180,E1 -12150.789,E2 -12150.789} C_VEL
LIN {X 0,Y 383.606,Z 564.759,A -85,B 0,C 180,E1 -12152.362,E2 -12152.362} C_VEL
LIN {X 0,Y 384.259,Z 557.09,A -85,B 0,C 180,E1 -12153.67,E2 -12153.67} C_VEL
LIN {X 0,Y 385.099,Z 546.683,A -85,B 0,C 180,E1 -12155.104,E2 -12155.104} C_VEL
LIN {X 0,Y 385.922,Z 536.094,A -85,B 0,C 180,E1 -12156.273,E2 -12156.273} C_VEL
LIN {X 0,Y 386.666,Z 525.845,A -85,B 0,C 180,E1 -12157.178,E2 -12157.178} C_VEL
LIN {X 0,Y 387.253,Z 513.648,A -85,B 0,C 180,E1 -12158.02,E2 -12158.02} C_VEL
LIN {X 0,Y 387.827,Z 500.792,A -85,B 0,C 180,E1 -12158.664,E2 -12158.664} C_VEL
LIN {X 0,Y 388.187,Z 488.677,A -85,B 0,C 180,E1 -12159.072,E2 -12159.072} C_VEL
LIN {X 0,Y 387.702,Z 482.91,A -85,B 0,C 180,E1 -12159.244,E2 -12159.244} C_VEL
LIN {X 0,Y 382.493,Z 464.165,A -85,B 0,C 180,E1 -12159.816,E2 -12159.816} C_VEL
LIN {X 0,Y 381.868,Z 458.348,A -85,B 0,C 180,E1 -12159.948,E2 -12159.948} C_VEL
LIN {X 0,Y 382.669,Z 404.357,A -85,B 0,C 180,E1 -12160.954,E2 -12160.954} C_VEL
LIN {X 0,Y 379.517,Z 389.12,A -85,B 0,C 180,E1 -12161.401,E2 -12161.401} C_VEL
LIN {X 0,Y 377.515,Z 382.309,A -85,B 0,C 180,E1 -12161.66,E2 -12161.66} C_VEL
LIN {X 0,Y 376.102,Z 374.638,A -85,B 0,C 180,E1 -12163.862,E2 -12163.862} C_VEL
LIN {X 0,Y 376.049,Z 374.639,A -85,B 0,C 180,E1 -12167.607,E2 -12167.607} C_VEL
LIN {X 0,Y 375.981,Z 374.65,A -85,B 0,C 180,E1 -12170.831,E2 -12170.831} C_VEL
LIN {X 0,Y 375.997,Z 374.651,A -85,B 0,C 180,E1 -12174.281,E2 -12174.281} C_VEL
LIN {X 0,Y 376.022,Z 374.647,A -85,B 0,C 180,E1 -12176.651,E2 -12176.651} C_VEL
LIN {X 0,Y 375.979,Z 374.649,A -85,B 0,C 180,E1 -12179.078,E2 -12179.078} C_VEL
LIN {X 0,Y 375.953,Z 374.654,A -85,B 0,C 180,E1 -12182.827,E2 -12182.827} C_VEL
LIN {X 0,Y 375.959,Z 374.651,A -85,B 0,C 180,E1 -12185.414,E2 -12185.414} C_VEL
LIN {X 0,Y 375.976,Z 374.654,A -85,B 0,C 180,E1 -12188.27,E2 -12188.27} C_VEL
LIN {X 0,Y 375.933,Z 374.654,A -85,B 0,C 180,E1 -12191.6,E2 -12191.6} C_VEL
LIN {X 0,Y 375.979,Z 374.648,A -85,B 0,C 180,E1 -12195.259,E2 -12195.259} C_VEL
LIN {X 0,Y 375.987,Z 374.652,A -85,B 0,C 180,E1 -12198.389,E2 -12198.389} C_VEL
LIN {X 0,Y 375.965,Z 374.653,A -85,B 0,C 180,E1 -12201.911,E2 -12201.911} C_VEL
LIN {X 0,Y 375.976,Z 374.649,A -85,B 0,C 180,E1 -12205.332,E2 -12205.332} C_VEL
LIN {X 0,Y 375.953,Z 374.656,A -85,B 0,C 180,E1 -12208.437,E2 -12208.437} C_VEL
LIN {X 0,Y 375.978,Z 374.654,A -85,B 0,C 180,E1 -12212.139,E2 -12212.139} C_VEL
LIN {X 0,Y 376.001,Z 374.649,A -85,B 0,C 180,E1 -12214.538,E2 -12214.538} C_VEL
LIN {X 0,Y 375.97,Z 374.655,A -85,B 0,C 180,E1 -12218.046,E2 -12218.046} C_VEL
LIN {X 0,Y 376.023,Z 374.644,A -85,B 0,C 180,E1 -12221.474,E2 -12221.474} C_VEL
LIN {X 0,Y 376.053,Z 374.64,A -85,B 0,C 180,E1 -12224.832,E2 -12224.832} C_VEL
LIN {X 0,Y 376.053,Z 374.644,A -85,B 0,C 180,E1 -12228.136,E2 -12228.136} C_VEL
LIN {X 0,Y 376.25,Z 374.619,A -85,B 0,C 180,E1 -12231.877,E2 -12231.877} C_VEL
LIN {X 0,Y 376.165,Z 374.627,A -85,B 0,C 180,E1 -12234.64,E2 -12234.64} C_VEL
LIN {X 0,Y 376.346,Z 374.607,A -85,B 0,C 180,E1 -12237.859,E2 -12237.859} C_VEL
LIN {X 0,Y 376.483,Z 374.591,A -85,B 0,C 180,E1 -12240,E2 -12240} C_VEL
LIN {X 0,Y 376.184,Z 374.623,A -85,B 0,C 180,E1 -12243.213,E2 -12243.213} C_VEL
LIN {X 0,Y 376.239,Z 374.619,A -85,B 0,C 180,E1 -12246.435,E2 -12246.435} C_VEL
LIN {X 0,Y 376.198,Z 374.623,A -85,B 0,C 180,E1 -12248.595,E2 -12248.595} C_VEL
LIN {X 0,Y 376.053,Z 374.644,A -85,B 0,C 180,E1 -12251.863,E2 -12251.863} C_VEL
LIN {X 0,Y 376.052,Z 374.64,A -85,B 0,C 180,E1 -12255.167,E2 -12255.167} C_VEL
LIN {X 0,Y 376.022,Z 374.645,A -85,B 0,C 180,E1 -12258.526,E2 -12258.526} C_VEL
LIN {X 0,Y 375.968,Z 374.655,A -85,B 0,C 180,E1 -12261.954,E2 -12261.954} C_VEL
LIN {X 0,Y 375.999,Z 374.647,A -85,B 0,C 180,E1 -12265.461,E2 -12265.461} C_VEL
LIN {X 0,Y 375.954,Z 374.652,A -85,B 0,C 180,E1 -12269.08,E2 -12269.08} C_VEL
LIN {X 0,Y 375.943,Z 374.653,A -85,B 0,C 180,E1 -12272.829,E2 -12272.829} C_VEL
LIN {X 0,Y 375.953,Z 374.653,A -85,B 0,C 180,E1 -12275.416,E2 -12275.416} C_VEL
LIN {X 0,Y 375.972,Z 374.652,A -85,B 0,C 180,E1 -12278.272,E2 -12278.272} C_VEL
LIN {X 0,Y 375.985,Z 374.651,A -85,B 0,C 180,E1 -12281.611,E2 -12281.611} C_VEL
LIN {X 0,Y 375.966,Z 374.651,A -85,B 0,C 180,E1 -12285.263,E2 -12285.263} C_VEL
LIN {X 0,Y 375.936,Z 374.654,A -85,B 0,C 180,E1 -12289.134,E2 -12289.134} C_VEL
LIN {X 0,Y 375.963,Z 374.656,A -85,B 0,C 180,E1 -12291.912,E2 -12291.912} C_VEL
LIN {X 0,Y 375.978,Z 374.65,A -85,B 0,C 180,E1 -12295.333,E2 -12295.333} C_VEL
LIN {X 0,Y 375.976,Z 374.649,A -85,B 0,C 180,E1 -12298.441,E2 -12298.441} C_VEL
LIN {X 0,Y 376.027,Z 374.772,A -85,B 0,C 180,E1 -12300.581,E2 -12300.581} C_VEL
LIN {X 0,Y 378.62,Z 387.401,A -85,B 0,C 180,E1 -12303.546,E2 -12303.546} C_VEL
LIN {X 0,Y 379.45,Z 392.894,A -85,B 0,C 180,E1 -12304.787,E2 -12304.787} C_VEL
LIN {X 0,Y 378.108,Z 408.953,A -85,B 0,C 180,E1 -12308.177,E2 -12308.177} C_VEL
LIN {X 0,Y 377.67,Z 414.649,A -85,B 0,C 180,E1 -12309.373,E2 -12309.373} C_VEL
LIN {X 0,Y 382.261,Z 448.566,A -85,B 0,C 180,E1 -12310.245,E2 -12310.245} C_VEL
LIN {X 0,Y 381.158,Z 523.367,A -85,B 0,C 180,E1 -12311.663,E2 -12311.663} C_VEL
LIN {X 0,Y 380.627,Z 536.656,A -85,B 0,C 180,E1 -12312.124,E2 -12312.124} C_VEL
LIN {X 0,Y 379.846,Z 549.409,A -85,B 0,C 180,E1 -12312.781,E2 -12312.781} C_VEL
LIN {X 0,Y 379.062,Z 560.74,A -85,B 0,C 180,E1 -12313.576,E2 -12313.576} C_VEL
LIN {X 0,Y 378.038,Z 572.447,A -85,B 0,C 180,E1 -12314.638,E2 -12314.638} C_VEL
LIN {X 0,Y 377.328,Z 582.329,A -85,B 0,C 180,E1 -12315.765,E2 -12315.765} C_VEL
LIN {X 0,Y 376.503,Z 591.609,A -85,B 0,C 180,E1 -12317.056,E2 -12317.056} C_VEL
LIN {X 0,Y 375.884,Z 599.548,A -85,B 0,C 180,E1 -12318.405,E2 -12318.405} C_VEL
LIN {X 0,Y 375.26,Z 607.282,A -85,B 0,C 180,E1 -12320.024,E2 -12320.024} C_VEL
LIN {X 0,Y 374.847,Z 614.415,A -85,B 0,C 180,E1 -12321.917,E2 -12321.917} C_VEL
LIN {X 0,Y 374.624,Z 619.144,A -85,B 0,C 180,E1 -12323.537,E2 -12323.537} C_VEL
LIN {X 0,Y 374.57,Z 622.747,A -85,B 0,C 180,E1 -12325.157,E2 -12325.157} C_VEL
LIN {X 0,Y 374.524,Z 625.322,A -85,B 0,C 180,E1 -12326.773,E2 -12326.773} C_VEL
LIN {X 0,Y 374.594,Z 626.532,A -85,B 0,C 180,E1 -12327.85,E2 -12327.85} C_VEL
LIN {X 0,Y 374.625,Z 627.292,A -85,B 0,C 180,E1 -12328.925,E2 -12328.925} C_VEL
LIN {X 0,Y 374.622,Z 627.618,A -85,B 0,C 180,E1 -12331.075,E2 -12331.075} C_VEL
LIN {X 0,Y 374.552,Z 627.198,A -85,B 0,C 180,E1 -12332.151,E2 -12332.151} C_VEL
LIN {X 0,Y 374.492,Z 626.348,A -85,B 0,C 180,E1 -12333.227,E2 -12333.227} C_VEL
LIN {X 0,Y 374.557,Z 625.091,A -85,B 0,C 180,E1 -12334.304,E2 -12334.304} C_VEL
LIN {X 0,Y 374.575,Z 622.166,A -85,B 0,C 180,E1 -12336.055,E2 -12336.055} C_VEL
LIN {X 0,Y 374.877,Z 617.327,A -85,B 0,C 180,E1 -12338.083,E2 -12338.083} C_VEL
LIN {X 0,Y 375.389,Z 611.17,A -85,B 0,C 180,E1 -12339.972,E2 -12339.972} C_VEL
LIN {X 0,Y 376.027,Z 604.477,A -85,B 0,C 180,E1 -12341.59,E2 -12341.59} C_VEL
LIN {X 0,Y 377.075,Z 596.198,A -85,B 0,C 180,E1 -12343.198,E2 -12343.198} C_VEL
LIN {X 0,Y 378.021,Z 586.601,A -85,B 0,C 180,E1 -12344.697,E2 -12344.697} C_VEL
LIN {X 0,Y 379.16,Z 576.133,A -85,B 0,C 180,E1 -12346.004,E2 -12346.004} C_VEL
LIN {X 0,Y 380.356,Z 565.592,A -85,B 0,C 180,E1 -12347.057,E2 -12347.057} C_VEL
LIN {X 0,Y 381.443,Z 553.906,A -85,B 0,C 180,E1 -12347.975,E2 -12347.975} C_VEL
LIN {X 0,Y 382.472,Z 541.782,A -85,B 0,C 180,E1 -12348.688,E2 -12348.688} C_VEL
LIN {X 0,Y 383.298,Z 528.582,A -85,B 0,C 180,E1 -12349.236,E2 -12349.236} C_VEL
LIN {X 0,Y 383.706,Z 515.431,A -85,B 0,C 180,E1 -12349.568,E2 -12349.568} C_VEL
LIN {X 0,Y 384.72,Z 447.691,A -85,B 0,C 180,E1 -12350.854,E2 -12350.854} C_VEL
LIN {X 0,Y 381.097,Z 425.451,A -85,B 0,C 180,E1 -12351.54,E2 -12351.54} C_VEL
LIN {X 0,Y 378.89,Z 414.179,A -85,B 0,C 180,E1 -12351.925,E2 -12351.925} C_VEL
LIN {X 0,Y 380.697,Z 396.77,A -85,B 0,C 180,E1 -12355.71,E2 -12355.71} C_VEL
LIN {X 0,Y 378.78,Z 386.428,A -85,B 0,C 180,E1 -12358.237,E2 -12358.237} C_VEL
LIN {X 0,Y 375.968,Z 374.65,A -85,B 0,C 180,E1 -12361.329,E2 -12361.329} C_VEL
LIN {X 0,Y 375.978,Z 374.653,A -85,B 0,C 180,E1 -12364.667,E2 -12364.667} C_VEL
LIN {X 0,Y 375.973,Z 374.652,A -85,B 0,C 180,E1 -12368.27,E2 -12368.27} C_VEL
LIN {X 0,Y 375.931,Z 374.657,A -85,B 0,C 180,E1 -12371.6,E2 -12371.6} C_VEL
LIN {X 0,Y 375.975,Z 374.648,A -85,B 0,C 180,E1 -12375.26,E2 -12375.26} C_VEL
LIN {X 0,Y 375.985,Z 374.645,A -85,B 0,C 180,E1 -12378.389,E2 -12378.389} C_VEL
LIN {X 0,Y 375.962,Z 374.651,A -85,B 0,C 180,E1 -12381.911,E2 -12381.911} C_VEL
LIN {X 0,Y 375.974,Z 374.652,A -85,B 0,C 180,E1 -12385.332,E2 -12385.332} C_VEL
LIN {X 0,Y 375.954,Z 374.652,A -85,B 0,C 180,E1 -12388.438,E2 -12388.438} C_VEL
LIN {X 0,Y 375.995,Z 374.646,A -85,B 0,C 180,E1 -12392.141,E2 -12392.141} C_VEL
LIN {X 0,Y 375.999,Z 374.63,A -85,B 0,C 180,E1 -12394.539,E2 -12394.539} C_VEL
LIN {X 0,Y 375.956,Z 374.652,A -85,B 0,C 180,E1 -12398.045,E2 -12398.045} C_VEL
LIN {X 0,Y 376.016,Z 374.645,A -85,B 0,C 180,E1 -12401.474,E2 -12401.474} C_VEL
LIN {X 0,Y 376.051,Z 374.638,A -85,B 0,C 180,E1 -12404.832,E2 -12404.832} C_VEL
LIN {X 0,Y 376.051,Z 374.639,A -85,B 0,C 180,E1 -12408.137,E2 -12408.137} C_VEL
LIN {X 0,Y 376.25,Z 374.616,A -85,B 0,C 180,E1 -12411.877,E2 -12411.877} C_VEL
LIN {X 0,Y 376.165,Z 374.621,A -85,B 0,C 180,E1 -12414.64,E2 -12414.64} C_VEL
LIN {X 0,Y 376.346,Z 374.6,A -85,B 0,C 180,E1 -12417.86,E2 -12417.86} C_VEL
LIN {X 0,Y 376.482,Z 374.584,A -85,B 0,C 180,E1 -12420,E2 -12420} C_VEL
LIN {X 0,Y 376.183,Z 374.619,A -85,B 0,C 180,E1 -12423.213,E2 -12423.213} C_VEL
LIN {X 0,Y 376.218,Z 374.62,A -85,B 0,C 180,E1 -12426.641,E2 -12426.641} C_VEL
LIN {X 0,Y 376.112,Z 374.632,A -85,B 0,C 180,E1 -12429.682,E2 -12429.682} C_VEL
LIN {X 0,Y 376.082,Z 374.634,A -85,B 0,C 180,E1 -12433.658,E2 -12433.658} C_VEL
LIN {X 0,Y 376.037,Z 374.638,A -85,B 0,C 180,E1 -12437.608,E2 -12437.608} C_VEL
LIN {X 0,Y 375.972,Z 374.648,A -85,B 0,C 180,E1 -12440.833,E2 -12440.833} C_VEL
LIN {X 0,Y 375.988,Z 374.646,A -85,B 0,C 180,E1 -12444.282,E2 -12444.282} C_VEL
LIN {X 0,Y 376.014,Z 374.629,A -85,B 0,C 180,E1 -12446.653,E2 -12446.653} C_VEL
LIN {X 0,Y 375.965,Z 374.651,A -85,B 0,C 180,E1 -12449.08,E2 -12449.08} C_VEL
LIN {X 0,Y 375.945,Z 374.655,A -85,B 0,C 180,E1 -12452.83,E2 -12452.83} C_VEL
LIN {X 0,Y 375.955,Z 374.654,A -85,B 0,C 180,E1 -12455.416,E2 -12455.416} C_VEL
LIN {X 0,Y 375.974,Z 374.654,A -85,B 0,C 180,E1 -12458.272,E2 -12458.272} C_VEL
LIN {X 0,Y 375.987,Z 374.651,A -85,B 0,C 180,E1 -12461.611,E2 -12461.611} C_VEL
LIN {X 0,Y 375.968,Z 374.657,A -85,B 0,C 180,E1 -12465.263,E2 -12465.263} C_VEL
LIN {X 0,Y 375.98,Z 374.654,A -85,B 0,C 180,E1 -12469.139,E2 -12469.139} C_VEL
LIN {X 0,Y 375.968,Z 374.655,A -85,B 0,C 180,E1 -12471.913,E2 -12471.913} C_VEL
LIN {X 0,Y 375.981,Z 374.651,A -85,B 0,C 180,E1 -12475.334,E2 -12475.334} C_VEL
LIN {X 0,Y 376.029,Z 374.721,A -85,B 0,C 180,E1 -12476.541,E2 -12476.541} C_VEL
LIN {X 0,Y 377.796,Z 382.953,A -85,B 0,C 180,E1 -12479.054,E2 -12479.054} C_VEL
LIN {X 0,Y 383.668,Z 398.064,A -85,B 0,C 180,E1 -12479.772,E2 -12479.772} C_VEL
LIN {X 0,Y 385.537,Z 406.381,A -85,B 0,C 180,E1 -12480.065,E2 -12480.065} C_VEL
LIN {X 0,Y 383.942,Z 489.596,A -85,B 0,C 180,E1 -12481.656,E2 -12481.656} C_VEL
LIN {X 0,Y 383.433,Z 502.231,A -85,B 0,C 180,E1 -12482.098,E2 -12482.098} C_VEL
LIN {X 0,Y 382.687,Z 514.711,A -85,B 0,C 180,E1 -12482.744,E2 -12482.744} C_VEL
LIN {X 0,Y 381.878,Z 525.495,A -85,B 0,C 180,E1 -12483.495,E2 -12483.495} C_VEL
LIN {X 0,Y 381.004,Z 536.682,A -85,B 0,C 180,E1 -12484.503,E2 -12484.503} C_VEL
LIN {X 0,Y 379.862,Z 547.24,A -85,B 0,C 180,E1 -12485.692,E2 -12485.692} C_VEL
LIN {X 0,Y 378.767,Z 557.05,A -85,B 0,C 180,E1 -12487.068,E2 -12487.068} C_VEL
LIN {X 0,Y 377.728,Z 565.916,A -85,B 0,C 180,E1 -12488.624,E2 -12488.624} C_VEL
LIN {X 0,Y 376.682,Z 573.88,A -85,B 0,C 180,E1 -12490.377,E2 -12490.377} C_VEL
LIN {X 0,Y 375.981,Z 580.004,A -85,B 0,C 180,E1 -12492.092,E2 -12492.092} C_VEL
LIN {X 0,Y 375.451,Z 584.465,A -85,B 0,C 180,E1 -12493.694,E2 -12493.694} C_VEL
LIN {X 0,Y 375.177,Z 586.896,A -85,B 0,C 180,E1 -12494.796,E2 -12494.796} C_VEL
LIN {X 0,Y 374.928,Z 588.872,A -85,B 0,C 180,E1 -12495.896,E2 -12495.896} C_VEL
LIN {X 0,Y 374.796,Z 590.639,A -85,B 0,C 180,E1 -12497.185,E2 -12497.185} C_VEL
LIN {X 0,Y 374.546,Z 592.2,A -85,B 0,C 180,E1 -12499.185,E2 -12499.185} C_VEL
LIN {X 0,Y 374.5,Z 592.395,A -85,B 0,C 180,E1 -12501.366,E2 -12501.366} C_VEL
LIN {X 0,Y 374.574,Z 591.863,A -85,B 0,C 180,E1 -12502.453,E2 -12502.453} C_VEL
LIN {X 0,Y 374.685,Z 590.666,A -85,B 0,C 180,E1 -12503.792,E2 -12503.792} C_VEL
LIN {X 0,Y 374.737,Z 587.898,A -85,B 0,C 180,E1 -12505.698,E2 -12505.698} C_VEL
LIN {X 0,Y 375.038,Z 584.449,A -85,B 0,C 180,E1 -12507.315,E2 -12507.315} C_VEL
LIN {X 0,Y 375.238,Z 579.941,A -85,B 0,C 180,E1 -12508.927,E2 -12508.927} C_VEL
LIN {X 0,Y 375.889,Z 573.086,A -85,B 0,C 180,E1 -12510.803,E2 -12510.803} C_VEL
LIN {X 0,Y 376.557,Z 565.682,A -85,B 0,C 180,E1 -12512.407,E2 -12512.407} C_VEL
LIN {X 0,Y 377.204,Z 558.139,A -85,B 0,C 180,E1 -12513.739,E2 -12513.739} C_VEL
LIN {X 0,Y 377.996,Z 548.999,A -85,B 0,C 180,E1 -12515.067,E2 -12515.067} C_VEL
LIN {X 0,Y 378.819,Z 538.827,A -85,B 0,C 180,E1 -12516.257,E2 -12516.257} C_VEL
LIN {X 0,Y 379.686,Z 527.548,A -85,B 0,C 180,E1 -12517.311,E2 -12517.311} C_VEL
LIN {X 0,Y 380.302,Z 515.884,A -85,B 0,C 180,E1 -12518.167,E2 -12518.167} C_VEL
LIN {X 0,Y 380.921,Z 503.008,A -85,B 0,C 180,E1 -12518.855,E2 -12518.855} C_VEL
LIN {X 0,Y 381.362,Z 489.232,A -85,B 0,C 180,E1 -12519.346,E2 -12519.346} C_VEL
LIN {X 0,Y 381.868,Z 458.348,A -85,B 0,C 180,E1 -12519.948,E2 -12519.948} C_VEL
LIN {X 0,Y 381.24,Z 452.536,A -85,B 0,C 180,E1 -12520.088,E2 -12520.088} C_VEL
LIN {X 0,Y 376.028,Z 433.807,A -85,B 0,C 180,E1 -12520.693,E2 -12520.693} C_VEL
LIN {X 0,Y 375.552,Z 427.994,A -85,B 0,C 180,E1 -12520.829,E2 -12520.829} C_VEL
LIN {X 0,Y 375.803,Z 404.848,A -85,B 0,C 180,E1 -12521.273,E2 -12521.273} C_VEL
LIN {X 0,Y 372.958,Z 391.114,A -85,B 0,C 180,E1 -12521.687,E2 -12521.687} C_VEL
LIN {X 0,Y 370.388,Z 382.732,A -85,B 0,C 180,E1 -12521.988,E2 -12521.988} C_VEL
LIN {X 0,Y 369.038,Z 375.52,A -85,B 0,C 180,E1 -12524.097,E2 -12524.097} C_VEL
LIN {X 0,Y 369.005,Z 375.517,A -85,B 0,C 180,E1 -12527.768,E2 -12527.768} C_VEL
LIN {X 0,Y 368.933,Z 375.526,A -85,B 0,C 180,E1 -12531.219,E2 -12531.219} C_VEL
LIN {X 0,Y 368.961,Z 375.525,A -85,B 0,C 180,E1 -12534.775,E2 -12534.775} C_VEL
LIN {X 0,Y 368.989,Z 375.525,A -85,B 0,C 180,E1 -12538.435,E2 -12538.435} C_VEL
LIN {X 0,Y 368.901,Z 375.535,A -85,B 0,C 180,E1 -12542.237,E2 -12542.237} C_VEL
LIN {X 0,Y 368.93,Z 375.527,A -85,B 0,C 180,E1 -12545.001,E2 -12545.001} C_VEL
LIN {X 0,Y 368.91,Z 375.532,A -85,B 0,C 180,E1 -12548.64,E2 -12548.64} C_VEL
LIN {X 0,Y 368.88,Z 375.535,A -85,B 0,C 180,E1 -12552.008,E2 -12552.008} C_VEL
LIN {X 0,Y 368.954,Z 375.523,A -85,B 0,C 180,E1 -12555.186,E2 -12555.186} C_VEL
LIN {X 0,Y 368.939,Z 375.53,A -85,B 0,C 180,E1 -12558.185,E2 -12558.185} C_VEL
LIN {X 0,Y 368.91,Z 375.529,A -85,B 0,C 180,E1 -12561.358,E2 -12561.358} C_VEL
LIN {X 0,Y 368.933,Z 375.526,A -85,B 0,C 180,E1 -12565.145,E2 -12565.145} C_VEL
LIN {X 0,Y 368.925,Z 375.527,A -85,B 0,C 180,E1 -12569.046,E2 -12569.046} C_VEL
LIN {X 0,Y 368.958,Z 375.524,A -85,B 0,C 180,E1 -12572.796,E2 -12572.796} C_VEL
LIN {X 0,Y 368.94,Z 375.531,A -85,B 0,C 180,E1 -12576.112,E2 -12576.112} C_VEL
LIN {X 0,Y 368.939,Z 375.529,A -85,B 0,C 180,E1 -12579.947,E2 -12579.947} C_VEL
LIN {X 0,Y 368.969,Z 375.522,A -85,B 0,C 180,E1 -12583.398,E2 -12583.398} C_VEL
LIN {X 0,Y 369.053,Z 375.512,A -85,B 0,C 180,E1 -12586.79,E2 -12586.79} C_VEL
LIN {X 0,Y 369.065,Z 375.515,A -85,B 0,C 180,E1 -12590.131,E2 -12590.131} C_VEL
LIN {X 0,Y 369.18,Z 375.5,A -85,B 0,C 180,E1 -12592.342,E2 -12592.342} C_VEL
LIN {X 0,Y 369.138,Z 375.503,A -85,B 0,C 180,E1 -12594.537,E2 -12594.537} C_VEL
LIN {X 0,Y 369.311,Z 375.482,A -85,B 0,C 180,E1 -12597.819,E2 -12597.819} C_VEL
LIN {X 0,Y 369.452,Z 375.467,A -85,B 0,C 180,E1 -12600,E2 -12600} C_VEL
LIN {X 0,Y 369.312,Z 375.484,A -85,B 0,C 180,E1 -12602.181,E2 -12602.181} C_VEL
LIN {X 0,Y 369.201,Z 375.495,A -85,B 0,C 180,E1 -12606.558,E2 -12606.558} C_VEL
LIN {X 0,Y 369.131,Z 375.502,A -85,B 0,C 180,E1 -12608.761,E2 -12608.761} C_VEL
LIN {X 0,Y 369.007,Z 375.522,A -85,B 0,C 180,E1 -12612.093,E2 -12612.093} C_VEL
LIN {X 0,Y 368.991,Z 375.52,A -85,B 0,C 180,E1 -12615.465,E2 -12615.465} C_VEL
LIN {X 0,Y 368.982,Z 375.52,A -85,B 0,C 180,E1 -12618.893,E2 -12618.893} C_VEL
LIN {X 0,Y 368.933,Z 375.528,A -85,B 0,C 180,E1 -12622.395,E2 -12622.395} C_VEL
LIN {X 0,Y 368.993,Z 375.524,A -85,B 0,C 180,E1 -12625.981,E2 -12625.981} C_VEL
LIN {X 0,Y 368.908,Z 375.533,A -85,B 0,C 180,E1 -12629.691,E2 -12629.691} C_VEL
LIN {X 0,Y 368.891,Z 375.531,A -85,B 0,C 180,E1 -12633.044,E2 -12633.044} C_VEL
LIN {X 0,Y 368.913,Z 375.532,A -85,B 0,C 180,E1 -12636.197,E2 -12636.197} C_VEL
LIN {X 0,Y 368.903,Z 375.53,A -85,B 0,C 180,E1 -12638.953,E2 -12638.953} C_VEL
LIN {X 0,Y 368.938,Z 375.53,A -85,B 0,C 180,E1 -12642.021,E2 -12642.021} C_VEL
LIN {X 0,Y 368.92,Z 375.528,A -85,B 0,C 180,E1 -12645.183,E2 -12645.183} C_VEL
LIN {X 0,Y 368.879,Z 375.536,A -85,B 0,C 180,E1 -12648.178,E2 -12648.178} C_VEL
LIN {X 0,Y 368.906,Z 375.531,A -85,B 0,C 180,E1 -12651.36,E2 -12651.36} C_VEL
LIN {X 0,Y 368.935,Z 375.526,A -85,B 0,C 180,E1 -12655.147,E2 -12655.147} C_VEL
LIN {X 0,Y 368.928,Z 375.527,A -85,B 0,C 180,E1 -12659.047,E2 -12659.047} C_VEL
LIN {X 0,Y 368.958,Z 375.685,A -85,B 0,C 180,E1 -12660.314,E2 -12660.314} C_VEL
LIN {X 0,Y 371.279,Z 386.768,A -85,B 0,C 180,E1 -12662.981,E2 -12662.981} C_VEL
LIN {X 0,Y 372.495,Z 394.118,A -85,B 0,C 180,E1 -12664.687,E2 -12664.687} C_VEL
LIN {X 0,Y 371.067,Z 410.139,A -85,B 0,C 180,E1 -12668.134,E2 -12668.134} C_VEL
LIN {X 0,Y 370.745,Z 414.247,A -85,B 0,C 180,E1 -12669.015,E2 -12669.015} C_VEL
LIN {X 0,Y 375.455,Z 448.446,A -85,B 0,C 180,E1 -12669.933,E2 -12669.933} C_VEL
LIN {X 0,Y 374.32,Z 523.539,A -85,B 0,C 180,E1 -12671.387,E2 -12671.387} C_VEL
LIN {X 0,Y 373.727,Z 537.429,A -85,B 0,C 180,E1 -12671.889,E2 -12671.889} C_VEL
LIN {X 0,Y 372.89,Z 550.369,A -85,B 0,C 180,E1 -12672.591,E2 -12672.591} C_VEL
LIN {X 0,Y 371.918,Z 562.977,A -85,B 0,C 180,E1 -12673.534,E2 -12673.534} C_VEL
LIN {X 0,Y 370.945,Z 574.22,A -85,B 0,C 180,E1 -12674.619,E2 -12674.619} C_VEL
LIN {X 0,Y 370.259,Z 583.329,A -85,B 0,C 180,E1 -12675.715,E2 -12675.715} C_VEL
LIN {X 0,Y 369.41,Z 592.651,A -85,B 0,C 180,E1 -12677.083,E2 -12677.083} C_VEL
LIN {X 0,Y 368.6,Z 601.705,A -85,B 0,C 180,E1 -12678.73,E2 -12678.73} C_VEL
LIN {X 0,Y 368.073,Z 608.994,A -85,B 0,C 180,E1 -12680.383,E2 -12680.383} C_VEL
LIN {X 0,Y 367.783,Z 613.908,A -85,B 0,C 180,E1 -12681.76,E2 -12681.76} C_VEL
LIN {X 0,Y 367.554,Z 618.676,A -85,B 0,C 180,E1 -12683.412,E2 -12683.412} C_VEL
LIN {X 0,Y 367.489,Z 622.314,A -85,B 0,C 180,E1 -12685.063,E2 -12685.063} C_VEL
LIN {X 0,Y 367.438,Z 624.92,A -85,B 0,C 180,E1 -12686.711,E2 -12686.711} C_VEL
LIN {X 0,Y 367.495,Z 626.148,A -85,B 0,C 180,E1 -12687.808,E2 -12687.808} C_VEL
LIN {X 0,Y 367.558,Z 626.937,A -85,B 0,C 180,E1 -12688.904,E2 -12688.904} C_VEL
LIN {X 0,Y 367.541,Z 627.308,A -85,B 0,C 180,E1 -12690,E2 -12690} C_VEL
LIN {X 0,Y 367.536,Z 627.292,A -85,B 0,C 180,E1 -12691.096,E2 -12691.096} C_VEL
LIN {X 0,Y 367.452,Z 626.886,A -85,B 0,C 180,E1 -12692.192,E2 -12692.192} C_VEL
LIN {X 0,Y 367.408,Z 626.066,A -85,B 0,C 180,E1 -12693.29,E2 -12693.29} C_VEL
LIN {X 0,Y 367.462,Z 624.823,A -85,B 0,C 180,E1 -12694.387,E2 -12694.387} C_VEL
LIN {X 0,Y 367.479,Z 622.241,A -85,B 0,C 180,E1 -12696.014,E2 -12696.014} C_VEL
LIN {X 0,Y 367.706,Z 618.567,A -85,B 0,C 180,E1 -12697.689,E2 -12697.689} C_VEL
LIN {X 0,Y 368.091,Z 613.841,A -85,B 0,C 180,E1 -12699.34,E2 -12699.34} C_VEL
LIN {X 0,Y 368.777,Z 606.76,A -85,B 0,C 180,E1 -12701.264,E2 -12701.264} C_VEL
LIN {X 0,Y 369.771,Z 599.117,A -85,B 0,C 180,E1 -12702.904,E2 -12702.904} C_VEL
LIN {X 0,Y 370.678,Z 591.317,A -85,B 0,C 180,E1 -12704.269,E2 -12704.269} C_VEL
LIN {X 0,Y 371.725,Z 581.819,A -85,B 0,C 180,E1 -12705.629,E2 -12705.629} C_VEL
LIN {X 0,Y 372.95,Z 571.313,A -85,B 0,C 180,E1 -12706.841,E2 -12706.841} C_VEL
LIN {X 0,Y 374.242,Z 559.632,A -85,B 0,C 180,E1 -12707.909,E2 -12707.909} C_VEL
LIN {X 0,Y 375.277,Z 548.294,A -85,B 0,C 180,E1 -12708.705,E2 -12708.705} C_VEL
LIN {X 0,Y 376.313,Z 534.81,A -85,B 0,C 180,E1 -12709.395,E2 -12709.395} C_VEL
LIN {X 0,Y 376.994,Z 521.554,A -85,B 0,C 180,E1 -12709.839,E2 -12709.839} C_VEL
LIN {X 0,Y 378.229,Z 448.681,A -85,B 0,C 180,E1 -12711.26,E2 -12711.26} C_VEL
LIN {X 0,Y 374.51,Z 425.859,A -85,B 0,C 180,E1 -12711.983,E2 -12711.983} C_VEL
LIN {X 0,Y 372.125,Z 413.718,A -85,B 0,C 180,E1 -12712.434,E2 -12712.434} C_VEL
LIN {X 0,Y 373.746,Z 399.316,A -85,B 0,C 180,E1 -12715.625,E2 -12715.625} C_VEL
LIN {X 0,Y 373.382,Z 395.429,A -85,B 0,C 180,E1 -12716.553,E2 -12716.553} C_VEL
LIN {X 0,Y 371.233,Z 385.152,A -85,B 0,C 180,E1 -12719.166,E2 -12719.166} C_VEL
LIN {X 0,Y 368.945,Z 375.528,A -85,B 0,C 180,E1 -12721.752,E2 -12721.752} C_VEL
LIN {X 0,Y 368.927,Z 375.531,A -85,B 0,C 180,E1 -12725.001,E2 -12725.001} C_VEL
LIN {X 0,Y 368.907,Z 375.53,A -85,B 0,C 180,E1 -12728.64,E2 -12728.64} C_VEL
LIN {X 0,Y 368.878,Z 375.534,A -85,B 0,C 180,E1 -12732.009,E2 -12732.009} C_VEL
LIN {X 0,Y 368.95,Z 375.522,A -85,B 0,C 180,E1 -12735.187,E2 -12735.187} C_VEL
LIN {X 0,Y 368.941,Z 375.523,A -85,B 0,C 180,E1 -12738.186,E2 -12738.186} C_VEL
LIN {X 0,Y 368.908,Z 375.53,A -85,B 0,C 180,E1 -12741.358,E2 -12741.358} C_VEL
LIN {X 0,Y 368.931,Z 375.528,A -85,B 0,C 180,E1 -12745.146,E2 -12745.146} C_VEL
LIN {X 0,Y 368.923,Z 375.53,A -85,B 0,C 180,E1 -12749.046,E2 -12749.046} C_VEL
LIN {X 0,Y 368.98,Z 375.525,A -85,B 0,C 180,E1 -12751.564,E2 -12751.564} C_VEL
LIN {X 0,Y 368.95,Z 375.506,A -85,B 0,C 180,E1 -12755.224,E2 -12755.224} C_VEL
LIN {X 0,Y 368.93,Z 375.53,A -85,B 0,C 180,E1 -12758.973,E2 -12758.973} C_VEL
LIN {X 0,Y 368.983,Z 375.52,A -85,B 0,C 180,E1 -12762.257,E2 -12762.257} C_VEL
LIN {X 0,Y 369.03,Z 375.513,A -85,B 0,C 180,E1 -12766.227,E2 -12766.227} C_VEL
LIN {X 0,Y 369.065,Z 375.506,A -85,B 0,C 180,E1 -12770.132,E2 -12770.132} C_VEL
LIN {X 0,Y 369.18,Z 375.497,A -85,B 0,C 180,E1 -12772.342,E2 -12772.342} C_VEL
LIN {X 0,Y 369.137,Z 375.496,A -85,B 0,C 180,E1 -12774.538,E2 -12774.538} C_VEL
LIN {X 0,Y 369.311,Z 375.477,A -85,B 0,C 180,E1 -12777.819,E2 -12777.819} C_VEL
LIN {X 0,Y 369.452,Z 375.46,A -85,B 0,C 180,E1 -12780,E2 -12780} C_VEL
LIN {X 0,Y 369.311,Z 375.48,A -85,B 0,C 180,E1 -12782.181,E2 -12782.181} C_VEL
LIN {X 0,Y 369.188,Z 375.498,A -85,B 0,C 180,E1 -12786.627,E2 -12786.627} C_VEL
LIN {X 0,Y 369.06,Z 375.51,A -85,B 0,C 180,E1 -12789.869,E2 -12789.869} C_VEL
LIN {X 0,Y 369.03,Z 375.513,A -85,B 0,C 180,E1 -12793.773,E2 -12793.773} C_VEL
LIN {X 0,Y 368.995,Z 375.516,A -85,B 0,C 180,E1 -12797.769,E2 -12797.769} C_VEL
LIN {X 0,Y 368.923,Z 375.525,A -85,B 0,C 180,E1 -12801.22,E2 -12801.22} C_VEL
LIN {X 0,Y 368.952,Z 375.517,A -85,B 0,C 180,E1 -12804.776,E2 -12804.776} C_VEL
LIN {X 0,Y 368.963,Z 375.511,A -85,B 0,C 180,E1 -12807.204,E2 -12807.204} C_VEL
LIN {X 0,Y 368.914,Z 375.531,A -85,B 0,C 180,E1 -12809.691,E2 -12809.691} C_VEL
LIN {X 0,Y 368.893,Z 375.532,A -85,B 0,C 180,E1 -12813.044,E2 -12813.044} C_VEL
LIN {X 0,Y 368.915,Z 375.532,A -85,B 0,C 180,E1 -12816.198,E2 -12816.198} C_VEL
LIN {X 0,Y 368.905,Z 375.531,A -85,B 0,C 180,E1 -12818.954,E2 -12818.954} C_VEL
LIN {X 0,Y 368.94,Z 375.525,A -85,B 0,C 180,E1 -12822.021,E2 -12822.021} C_VEL
LIN {X 0,Y 368.922,Z 375.535,A -85,B 0,C 180,E1 -12825.184,E2 -12825.184} C_VEL
LIN {X 0,Y 368.909,Z 375.537,A -85,B 0,C 180,E1 -12828.182,E2 -12828.182} C_VEL
LIN {X 0,Y 368.913,Z 375.533,A -85,B 0,C 180,E1 -12831.36,E2 -12831.36} C_VEL
LIN {X 0,Y 368.938,Z 375.529,A -85,B 0,C 180,E1 -12835.148,E2 -12835.148} C_VEL
LIN {X 0,Y 368.983,Z 375.643,A -85,B 0,C 180,E1 -12836.144,E2 -12836.144} C_VEL
LIN {X 0,Y 370.606,Z 383.268,A -85,B 0,C 180,E1 -12838.531,E2 -12838.531} C_VEL
LIN {X 0,Y 377.335,Z 399.871,A -85,B 0,C 180,E1 -12839.37,E2 -12839.37} C_VEL
LIN {X 0,Y 379.047,Z 407.244,A -85,B 0,C 180,E1 -12839.641,E2 -12839.641} C_VEL
LIN {X 0,Y 377.407,Z 489.905,A -85,B 0,C 180,E1 -12841.249,E2 -12841.249} C_VEL
LIN {X 0,Y 376.923,Z 501.73,A -85,B 0,C 180,E1 -12841.662,E2 -12841.662} C_VEL
LIN {X 0,Y 376.148,Z 514.215,A -85,B 0,C 180,E1 -12842.305,E2 -12842.305} C_VEL
LIN {X 0,Y 375.219,Z 526.08,A -85,B 0,C 180,E1 -12843.137,E2 -12843.137} C_VEL
LIN {X 0,Y 374.196,Z 538.12,A -85,B 0,C 180,E1 -12844.258,E2 -12844.258} C_VEL
LIN {X 0,Y 372.974,Z 548.813,A -85,B 0,C 180,E1 -12845.51,E2 -12845.51} C_VEL
LIN {X 0,Y 371.842,Z 558.372,A -85,B 0,C 180,E1 -12846.91,E2 -12846.91} C_VEL
LIN {X 0,Y 370.671,Z 567.639,A -85,B 0,C 180,E1 -12848.617,E2 -12848.617} C_VEL
LIN {X 0,Y 369.681,Z 574.855,A -85,B 0,C 180,E1 -12850.279,E2 -12850.279} C_VEL
LIN {X 0,Y 369.056,Z 579.76,A -85,B 0,C 180,E1 -12851.687,E2 -12851.687} C_VEL
LIN {X 0,Y 368.486,Z 584.49,A -85,B 0,C 180,E1 -12853.376,E2 -12853.376} C_VEL
LIN {X 0,Y 368.047,Z 588.067,A -85,B 0,C 180,E1 -12855.062,E2 -12855.062} C_VEL
LIN {X 0,Y 367.743,Z 590.994,A -85,B 0,C 180,E1 -12857.079,E2 -12857.079} C_VEL
LIN {X 0,Y 367.477,Z 592.484,A -85,B 0,C 180,E1 -12858.975,E2 -12858.975} C_VEL
LIN {X 0,Y 367.416,Z 592.749,A -85,B 0,C 180,E1 -12861.198,E2 -12861.198} C_VEL
LIN {X 0,Y 367.482,Z 592.286,A -85,B 0,C 180,E1 -12862.307,E2 -12862.307} C_VEL
LIN {X 0,Y 367.607,Z 590.987,A -85,B 0,C 180,E1 -12863.805,E2 -12863.805} C_VEL
LIN {X 0,Y 367.715,Z 587.406,A -85,B 0,C 180,E1 -12866.164,E2 -12866.164} C_VEL
LIN {X 0,Y 368.023,Z 583.688,A -85,B 0,C 180,E1 -12867.811,E2 -12867.811} C_VEL
LIN {X 0,Y 368.285,Z 578.878,A -85,B 0,C 180,E1 -12869.453,E2 -12869.453} C_VEL
LIN {X 0,Y 368.906,Z 572.796,A -85,B 0,C 180,E1 -12871.092,E2 -12871.092} C_VEL
LIN {X 0,Y 369.625,Z 565.253,A -85,B 0,C 180,E1 -12872.724,E2 -12872.724} C_VEL
LIN {X 0,Y 370.447,Z 555.787,A -85,B 0,C 180,E1 -12874.352,E2 -12874.352} C_VEL
LIN {X 0,Y 371.352,Z 546.016,A -85,B 0,C 180,E1 -12875.702,E2 -12875.702} C_VEL
LIN {X 0,Y 372.253,Z 535.071,A -85,B 0,C 180,E1 -12876.913,E2 -12876.913} C_VEL
LIN {X 0,Y 373.166,Z 522.606,A -85,B 0,C 180,E1 -12877.984,E2 -12877.984} C_VEL
LIN {X 0,Y 373.773,Z 510.336,A -85,B 0,C 180,E1 -12878.787,E2 -12878.787} C_VEL
LIN {X 0,Y 374.327,Z 497.228,A -85,B 0,C 180,E1 -12879.387,E2 -12879.387} C_VEL
LIN {X 0,Y 374.66,Z 484.703,A -85,B 0,C 180,E1 -12879.75,E2 -12879.75} C_VEL
LIN {X 0,Y 375.552,Z 427.994,A -85,B 0,C 180,E1 -12880.829,E2 -12880.829} C_VEL
LIN {X 0,Y 375.115,Z 422.155,A -85,B 0,C 180,E1 -12880.965,E2 -12880.965} C_VEL
LIN {X 0,Y 373.756,Z 416.476,A -85,B 0,C 180,E1 -12881.143,E2 -12881.143} C_VEL
LIN {X 0,Y 369.84,Z 405.398,A -85,B 0,C 180,E1 -12881.558,E2 -12881.558} C_VEL
LIN {X 0,Y 367.573,Z 397.862,A -85,B 0,C 180,E1 -12881.824,E2 -12881.824} C_VEL
LIN {X 0,Y 364.57,Z 387.119,A -85,B 0,C 180,E1 -12882.199,E2 -12882.199} C_VEL
LIN {X 0,Y 363.274,Z 383.036,A -85,B 0,C 180,E1 -12882.358,E2 -12882.358} C_VEL
LIN {X 0,Y 361.994,Z 376.397,A -85,B 0,C 180,E1 -12884.334,E2 -12884.334} C_VEL
LIN {X 0,Y 361.964,Z 376.396,A -85,B 0,C 180,E1 -12888.099,E2 -12888.099} C_VEL
LIN {X 0,Y 361.896,Z 376.402,A -85,B 0,C 180,E1 -12891.652,E2 -12891.652} C_VEL
LIN {X 0,Y 361.931,Z 376.398,A -85,B 0,C 180,E1 -12895.289,E2 -12895.289} C_VEL
LIN {X 0,Y 361.925,Z 376.399,A -85,B 0,C 180,E1 -12897.777,E2 -12897.777} C_VEL
LIN {X 0,Y 361.848,Z 376.408,A -85,B 0,C 180,E1 -12901.284,E2 -12901.284} C_VEL
LIN {X 0,Y 361.856,Z 376.413,A -85,B 0,C 180,E1 -12904.279,E2 -12904.279} C_VEL
LIN {X 0,Y 361.865,Z 376.406,A -85,B 0,C 180,E1 -12907.222,E2 -12907.222} C_VEL
LIN {X 0,Y 361.835,Z 376.412,A -85,B 0,C 180,E1 -12910.754,E2 -12910.754} C_VEL
LIN {X 0,Y 361.861,Z 376.413,A -85,B 0,C 180,E1 -12914.36,E2 -12914.36} C_VEL
LIN {X 0,Y 361.882,Z 376.404,A -85,B 0,C 180,E1 -12917.559,E2 -12917.559} C_VEL
LIN {X 0,Y 361.872,Z 376.406,A -85,B 0,C 180,E1 -12920.971,E2 -12920.971} C_VEL
LIN {X 0,Y 361.871,Z 376.408,A -85,B 0,C 180,E1 -12924.654,E2 -12924.654} C_VEL
LIN {X 0,Y 361.833,Z 376.416,A -85,B 0,C 180,E1 -12928.37,E2 -12928.37} C_VEL
LIN {X 0,Y 361.903,Z 376.407,A -85,B 0,C 180,E1 -12932.22,E2 -12932.22} C_VEL
LIN {X 0,Y 361.923,Z 376.401,A -85,B 0,C 180,E1 -12934.709,E2 -12934.709} C_VEL
LIN {X 0,Y 361.895,Z 376.408,A -85,B 0,C 180,E1 -12938.347,E2 -12938.347} C_VEL
LIN {X 0,Y 361.962,Z 376.399,A -85,B 0,C 180,E1 -12942.06,E2 -12942.06} C_VEL
LIN {X 0,Y 361.992,Z 376.396,A -85,B 0,C 180,E1 -12946.1,E2 -12946.1} C_VEL
LIN {X 0,Y 362.029,Z 376.39,A -85,B 0,C 180,E1 -12949.938,E2 -12949.938} C_VEL
LIN {X 0,Y 362.144,Z 376.377,A -85,B 0,C 180,E1 -12952.192,E2 -12952.192} C_VEL
LIN {X 0,Y 362.111,Z 376.379,A -85,B 0,C 180,E1 -12954.431,E2 -12954.431} C_VEL
LIN {X 0,Y 362.276,Z 376.358,A -85,B 0,C 180,E1 -12957.776,E2 -12957.776} C_VEL
LIN {X 0,Y 362.422,Z 376.342,A -85,B 0,C 180,E1 -12960,E2 -12960} C_VEL
LIN {X 0,Y 362.276,Z 376.36,A -85,B 0,C 180,E1 -12962.223,E2 -12962.223} C_VEL
LIN {X 0,Y 362.164,Z 376.37,A -85,B 0,C 180,E1 -12966.686,E2 -12966.686} C_VEL
LIN {X 0,Y 362.068,Z 376.381,A -85,B 0,C 180,E1 -12968.933,E2 -12968.933} C_VEL
LIN {X 0,Y 361.96,Z 376.398,A -85,B 0,C 180,E1 -12972.332,E2 -12972.332} C_VEL
LIN {X 0,Y 361.955,Z 376.396,A -85,B 0,C 180,E1 -12974.62,E2 -12974.62} C_VEL
LIN {X 0,Y 361.954,Z 376.401,A -85,B 0,C 180,E1 -12978.099,E2 -12978.099} C_VEL
LIN {X 0,Y 361.893,Z 376.406,A -85,B 0,C 180,E1 -12981.653,E2 -12981.653} C_VEL
LIN {X 0,Y 361.921,Z 376.4,A -85,B 0,C 180,E1 -12985.29,E2 -12985.29} C_VEL
LIN {X 0,Y 361.901,Z 376.406,A -85,B 0,C 180,E1 -12987.779,E2 -12987.779} C_VEL
LIN {X 0,Y 361.831,Z 376.413,A -85,B 0,C 180,E1 -12991.63,E2 -12991.63} C_VEL
LIN {X 0,Y 361.869,Z 376.407,A -85,B 0,C 180,E1 -12995.345,E2 -12995.345} C_VEL
LIN {X 0,Y 361.87,Z 376.406,A -85,B 0,C 180,E1 -12999.028,E2 -12999.028} C_VEL
LIN {X 0,Y 361.88,Z 376.406,A -85,B 0,C 180,E1 -13002.441,E2 -13002.441} C_VEL
LIN {X 0,Y 361.843,Z 376.413,A -85,B 0,C 180,E1 -13005.637,E2 -13005.637} C_VEL
LIN {X 0,Y 361.832,Z 376.411,A -85,B 0,C 180,E1 -13009.245,E2 -13009.245} C_VEL
LIN {X 0,Y 361.862,Z 376.406,A -85,B 0,C 180,E1 -13012.778,E2 -13012.778} C_VEL
LIN {X 0,Y 361.854,Z 376.413,A -85,B 0,C 180,E1 -13015.721,E2 -13015.721} C_VEL
LIN {X 0,Y 361.919,Z 376.404,A -85,B 0,C 180,E1 -13019.677,E2 -13019.677} C_VEL
LIN {X 0,Y 361.944,Z 376.607,A -85,B 0,C 180,E1 -13020.049,E2 -13020.049} C_VEL
LIN {X 0,Y 364.488,Z 388.981,A -85,B 0,C 180,E1 -13023.081,E2 -13023.081} C_VEL
LIN {X 0,Y 365.509,Z 395.638,A -85,B 0,C 180,E1 -13024.651,E2 -13024.651} C_VEL
LIN {X 0,Y 364.045,Z 411.097,A -85,B 0,C 180,E1 -13028.042,E2 -13028.042} C_VEL
LIN {X 0,Y 363.838,Z 413.948,A -85,B 0,C 180,E1 -13028.665,E2 -13028.665} C_VEL
